- Модуль ВЧ-демпфування: Несправність: перенапруга 24 В'; 37052 'F37052 - Модуль ВЧ-демпфування: Помилка даних EEPROM'; 37056 'A37056 (F) - Модуль ВЧ-демпфування: Перегрів радіатора'; 37310 'A37310 (F) - Модуль ВЧ-дроселя: Перегрів'; 37311 'F37311 - Модуль ВЧ-дроселя: Перегрів радіатора'; 37312 'A37312 (F) - Модуль ВЧ-дроселя: Перегрів або несправність вентилятора'; 37313 'F37313 - Модуль ВЧ-дроселя: Перегрів або несправність вентилятора'; 37502 'A37502 (F) - Модуль ВЧ-демпфування: Напруга демпфування занадто висока'; 37800 'N37800 (F) - Модуль ВЧ-демпфування: Груповий сигнал'; 37801 'A37801 (F, N) - Модуль ВЧ-демпфування: Відсутній сигнал справності'; 37802 'F37802 (N, A) - Модуль ВЧ-демпфування: Переповнення часового кванта'; 37804 'F37804 (N, A) - Модуль ВЧ-демпфування: CRC'; 37805 'F37805 - Модуль ВЧ-демпфування: Некоректна контрольна сума EEPROM'; 37820 'F37820 - Модуль ВЧ-демпфування: Помилка телеграми'; 37835 'F37835 - Модуль ВЧ-демпфування: Помилка циклічної передачі даних'; 37836 'F37836 - Модуль ВЧ-демпфування: Помилка передавання даних DRIVE-CLiQ'; 37837 'F37837 - Модуль ВЧ-демпфування: Несправність компонента'; 37845 'F37845 - Модуль ВЧ-демпфування: Помилка циклічної передачі даних'; 37850 'F37850 - Модуль ВЧ-демпфування: Внутрішня програмна помилка'; 37851 'F37851 - Модуль ВЧ-демпфування (CU): Відсутній сигнал справності'; 37860 'F37860 - Модуль ВЧ-демпфування (CU): Помилка телеграми'; 37875 'F37875 - Модуль ВЧ-демпфування: Несправність напруги живлення'; 37885 'F37885 - Модуль ВЧ-демпфування (CU): Помилка циклічної передачі даних'; 37886 'F37886 - Модуль ВЧ-демпфування (CU): Помилка під час передавання даних DRIVE-CLiQ'; 37887 'F37887 - Модуль ВЧ-демпфування (CU): Несправність компонента'; 37895 'F37895 - Модуль ВЧ-демпфування (CU): Помилка почергової циклічної передачі даних'; 37896 'F37896 - Модуль ВЧ-демпфування (CU): Некоректні властивості компонента'; 37899 'F37899 (N, A) - Модуль ВЧ-демпфування: Невідома несправність'; 37903 'F37903 - Модуль ВЧ-демпфування: Виникла помилка I2C-шини'; 37950 'F37950 - Модуль ВЧ-демпфування: Внутрішня програмна помилка'; 37999 'A37999 (F, N) - Модуль ВЧ-демпфування: Невідоме аварійне повідомлення'; 40000 'F40000 - Несправність роз’єму DRIVE-CLiQ X100'; 40001 'F40001 - Несправність роз’єму DRIVE-CLiQ X101'; 40002 'F40002 - Несправність роз’єму DRIVE-CLiQ X102'; 40003 'F40003 - Несправність роз’єму DRIVE-CLiQ X103'; 40004 'F40004 - Несправність роз’єму DRIVE-CLiQ X104'; 40005 'F40005 - Несправність роз’єму DRIVE-CLiQ X105'; 40100 'A40100 - Аварійне повідомлення роз’єму DRIVE-CLiQ X100'; 40101 'A40101 - Аварійне повідомлення роз’єму DRIVE-CLiQ X101'; 40102 'A40102 - Аварійне повідомлення роз’єму DRIVE-CLiQ X102'; 40103 'A40103 - Аварійне повідомлення роз’єму DRIVE-CLiQ X103'; 40104 'A40104 - Аварійне повідомлення роз’єму DRIVE-CLiQ X104'; 40105 'A40105 - Аварійне повідомлення роз’єму DRIVE-CLiQ X105'; 40799 'F40799 - CX32: Перевищено налаштований час завершення передавання'; 40801 'F40801 - CX32 DRIVE-CLiQ: відсутній сигнал справності'; 40820 'F40820 - CX32 DRIVE-CLiQ: помилка телеграми'; 40825 'F40825 - CX32 DRIVE-CLiQ: Несправність напруги живлення'; 40835 'F40835 - CX32 DRIVE-CLiQ: помилка циклічної передачі даних'; 40836 'F40836 - CX32 DRIVE-CLiQ: помилка передавання даних DRIVE-CLiQ'; 40837 'F40837 - CX32 DRIVE-CLiQ: несправність компонента'; 40845 'F40845 - CX32 DRIVE-CLiQ: помилка циклічної передачі даних'; 40851 'F40851 - CX32 DRIVE-CLiQ (CU): відсутній сигнал справності'; 40860 'F40860 - CX32 DRIVE-CLiQ (CU): помилка телеграми'; 40875 'F40875 - CX32 DRIVE-CLiQ (CU): Несправність напруги живлення'; 40885 'F40885 - CX32 DRIVE-CLiQ (CU): помилка циклічної передачі даних'; 40886 'F40886 - CX32 DRIVE-CLiQ (CU): помилка під час передавання даних DRIVE-CLiQ'; 40887 'F40887 - CX32 DRIVE-CLiQ (CU): несправність компонента'; 40895 'F40895 - CX32 DRIVE-CLiQ (CU): помилка циклічної передачі даних'; 49150 'F49150 - Охолоджувальний агрегат: Виникла несправність'; 49151 'F49151 - Охолоджувальний агрегат: Провідність перевищила поріг несправності'; 49152 'F49152 - Охолоджувальний агрегат: Відсутній сигнал зворотного зв’язку команди ON'; 49153 'F49153 - Охолоджувальний агрегат: Витрата рідини занадто мала'; 49154 'F49154 (A) - Охолоджувальний агрегат: Виявлено витік рідини'; 49155 'F49155 - Охолоджувальний агрегат: Адаптер Power Stack: версія прошивки застаріла'; 49156 'F49156 - Охолоджувальний агрегат: Температура охолоджувальної рідини перевищила поріг несправності'; 49170 'A49170 - Охолоджувальний агрегат: Виникло аварійне повідомлення'; 49171 'A49171 (N) - Охолоджувальний агрегат: Провідність перевищила поріг аварійного повідомлення'; 49172 'A49172 - Охолоджувальний агрегат: Фактичне значення провідності некоректне'; 49173 'A49173 - Охолоджувальний агрегат: Температура охолоджувальної рідини перевищила поріг аварійного повідомлення'; 49200 'F49200 - Несправність групового сигналу збудження'; 49201 'A49201 (F) - Аварійне повідомлення групового сигналу збудження'; 49204 'A49204 (N) - Аварійне повідомлення про вимкнення збудження'; 49205 'A49205 - Збудження: некоректна параметризація безщіткового збуджувача'; 49920 'A49920 (F) - Спрацював захисний автомат головного кола'; 49921 'A49921 (F) - Спрацював захисний автомат резервного головного кола'; 49922 'A49922 (F) - Спрацював захисний автомат кола 24 В'; 49923 'A49923 (F) - Спрацював захисний автомат кола 24 В клемної колодки'; 49924 'A49924 (F) - Спрацював захисний автомат кола живлення силового модуля'; 49926 'A49926 (F) - Спрацював захисний автомат кола синхронізувальної напруги'; 49927 'A49927 (F) - Спрацював захисний автомат кола допоміжного вентилятора'; 49933 'A49933 (F) - Спрацював захисний автомат кола збудження 230 В AC'; 49934 'A49934 (F) - Спрацював захисний автомат вихідного кола охолоджувального агрегату 230 В AC'; 49935 'A49935 (F) - Спрацював захисний автомат кола 24 В соленоїдів дверей силового модуля'; 49936 'A49936 - Спрацював захисний автомат кола освітлення/розеток 230 В AC'; 49937 'A49937 (F) - UPS не готовий до роботи'; 49938 'A49938 (F) - Робота від батареї UPS'; 49939 'A49939 (F) - Батарею UPS розряджено'; 49940 'A49940 (F) - Спрацював захисний автомат кола живлення силового модуля 400 В'; 49941 'A49941 (F) - Спрацював захисний автомат антиконденсаційного обігріву'; 49942 'A49942 (F) - Спрацював захисний автомат кола живлення SITOP'; 49998 'A49998 - Виникла подія запуску реєстратора'; 50002 'A50002 (F) - COMM BOARD: аварійне повідомлення 2'; 50003 'A50003 (F) - COMM BOARD: аварійне повідомлення 3'; 50004 'A50004 (F) - COMM BOARD: аварійне повідомлення 4'; 50005 'A50005 (F) - COMM BOARD: аварійне повідомлення 5'; 50006 'A50006 (F) - COMM BOARD: аварійне повідомлення 6'; 50007 'A50007 (F) - COMM BOARD: аварійне повідомлення 7'; 50008 'A50008 (F) - COMM BOARD: аварійне повідомлення 8'; 50011 'A50011 (F) - EtherNetIP/COMM BOARD: помилка конфігурації'; 0 'Немає попередження'

text list "LiftUpStatus": 0 'Не має статусу'; 1 'Рухається вверх'; 2 'Рухається вниз'; 4 'Зупинено і Готовий до роботи (в середній зоні)'; 8 'Зупинено і НЕ готовий до роботи'; 16 'Аварія'; 32 'Зупинено у верхньому положенні'; 64 'Зупинено у нижньому положенні'

text list "TrolleyStatus": 1 'Рухається вперед'; 2 'Рухається назад'; 4 'Зупинено і Готовий до роботи'; 8 'Зупинено і НЕ готовий до роботи'; 16 'Аварія візка'; 32 'Зупинено у крайньому положенні Вперед'; 64 'Зупинено у крайньому положенні Назад'; 0 'Не має статусу'

text list "CraneStatus": 0 'Не має статусу'; 1 'Рухається вліво'; 2 'Рухається вправо'; 4 'Зупинено і Готовий до роботи'; 8 'Зупинено і НЕ готовий до роботи'; 16 'Аварія візка'; 32 'Зупинено у крайньому положенні Вліво'; 64 'Зупинено у крайньому положенні Вправо'

text list "LiftUpCondition": 0 'Очікується запуск калібровки'; 10 'Відпустіть всі кнопки керування / Відпустіть кнопки керування'; 20 'Натисніть кнопку «Підйом»'; 30 'Досягніть реперної точки 1K1'; 40 'Відпустіть кнопку «Підйом»'; 50 'Натисніть кноп. «Опускання», звільнить 1К1 та відпустіть кноп. / Звільніть 1K1 та відпустіть кнопку «Опускання»'; 60 'Відхід завершено'; 70 'Натисніть кнопку «Підйом»'; 80 'Повторно досягніть 1K1 та відпустіть кнопку / Повторно досягніть реперної точки 1K1'; 90 'Виконується Quick Stop'; 100 'Очікується повна зупинка привода, відпустіть кнопку "Підйом" / Очікується повна зупинка привода'; 110 'Запускається preset енкодера'; 120 'Очікується підтвердження preset енкодера / Очікується підтвердження preset'; 130 'Калібровка завершена'; 900 'Процедуру перервано'; 910 'Процедура завершена з помилкою'; 5 'Опустіться до звільнення 1К1 та відпустіть кнопку'

text list "LiftUpStepName": 0 'Калібровка неактивна'; 10 'Перевірка умов калібровки'; 20 'Очікування команди підйому'; 30 'Перший підхід до реперної точки'; 40 'Перше проходження 1K1'; 50 'Відхід нижче реперної точки'; 60 'Відхід завершено'; 70 'Очікування повторного підйому'; 80 'Повторний підхід до реперної точки'; 90 'Quick Stop'; 100 'Очікування зупинки привода'; 110 'Запуск preset енкодера'; 120 'Очікування завершення preset'; 130 'Калібровку успішно завершено'; 900 'Калібровку перервано'; 910 'Помилка калібровки'; 5 'Попередній відхід від реперної точки'

text list "TrolleyCondition": 0 'Очікується запуск калібровки'; 5 'Опустіться до звільнення 3К1 та відпустіть кнопку "Назад"'; 10 'Відпустіть всі кнопки керування / Відпустіть кнопки керування'; 20 'Натисніть кнопку «Підйом» / Натисніть кнопку «Вперед»'; 30 'Досягніть реперної точки 1K1 / Досягніть реперної точки 3K1'; 40 'Відпустіть кнопку «Підйом» / Відпустіть кнопку «Вперед»'; 50 'Звільніть 1K1 та відпустіть кнопку «Опускання» / Звільніть 3K1 та відпустіть кнопку «Назад»'; 60 'Відхід завершено'; 70 'Натисніть кнопку «Підйом» / Натисніть кнопку «Вперед»'; 80 'Повторно досягніть реперної точки 1K1 / Повторно досягніть 3K1 та відпустіть кнопку'; 90 'Виконується Quick Stop'; 100 'Очікується повна зупинка привода / Очікується повна зупинка привода, відпустіть кнопку "Вперед"'; 110 'Запускається preset енкодера'; 120 'Очікується підтвердження preset енкодера / Очікується підтвердження preset'; 130 'Калібровка завершена'; 900 'Процедуру перервано'; 910 'Процедура завершена з помилкою'

text list "TrolleyStepName": 0 'Калібровка неактивна'; 5 'Попередній відхід від реперної точки'; 10 'Перевірка умов калібровки'; 20 'Очікування команди підйому / Очікування команди руху вперед'; 30 'Перший підхід до реперної точки'; 40 'Перше проходження 1K1 / Перше проходження 3K1'; 50 'Відхід нижче реперної точки / Відхід назад від реперної точки'; 60 'Відхід завершено'; 70 'Очікування повторного підйому / Очікування повторного руху вперед'; 80 'Повторний підхід до реперної точки'; 90 'Quick Stop'; 100 'Очікування зупинки привода'; 110 'Запуск preset енкодера'; 120 'Очікування завершення preset'; 130 'Калібровку успішно завершено'; 900 'Калібровку перервано'; 910 'Помилка калібровки'

text list "CraneCondition": 0 'Очікується запуск калібровки'; 5 'Очікується звільнення 4К1 та відпустіть кнопку "Вправо"'; 10 'Відпустіть всі кнопки керування / Відпустіть кнопки керування'; 20 'Натисніть кнопку «Підйом» / Натисніть кнопку «Вліво»'; 30 'Досягніть реперної точки 1K1 / Досягніть реперної точки 4K1'; 40 'Відпустіть кнопку «Підйом» / Відпустіть кнопку «Вліво»'; 50 'Звільніть 1K1 та відпустіть кнопку «Опускання» / Звільніть 4K1 та відпустіть кнопку «Вправо»'; 60 'Відхід завершено'; 70 'Натисніть кнопку «Підйом» / Натисніть кнопку «Вліво»'; 80 'Повторно досягніть реперної точки 1K1 / Повторно досягніть 4K1 та відпустіть кнопку'; 90 'Виконується Quick Stop'; 100 'Очікується повна зупинка привода / Очікується повна зупинка обох приводів, відпустіть кнопку "Вліво"'; 110 'Запускається preset енкодера'; 120 'Очікується підтвердження preset / Очікується підтвердження preset обох енкодерів'; 130 'Калібровка завершена'; 900 'Процедуру перервано'; 910 'Процедура завершена з помилкою'

text list "CraneStepName": 0 'Калібровка неактивна'; 5 'Попередній відхід від реперної точки'; 10 'Перевірка умов калібровки'; 20 'Очікування команди підйому / Очікування команди руху вліво'; 30 'Перший підхід до реперної точки'; 40 'Перше проходження 1K1 / Перше проходження 4K1'; 50 'Відхід нижче реперної точки / Відхід вправо від реперної точки'; 60 'Відхід завершено'; 70 'Очікування повторного підйому / Очікування повторного руху вліво'; 80 'Повторний підхід до реперної точки'; 90 'Quick Stop'; 100 'Очікування зупинки привода / Очікування зупинки приводів'; 110 'Запуск preset енкодера / Запуск preset енкодерів'; 120 'Очікування завершення preset'; 130 'Калібровку успішно завершено'; 900 'Калібровку перервано'; 910 'Помилка калібровки'

Template "Template_1" 800x454
   Button "btnSettings" at 620,411 size 83x40; TextOff 'Exit'; PictureOn "ExitRuntime_TP700_Comfort_TR"; PictureOff "Navigates to System screens for TP700 Comfort 17.0.0.0"; Authorization "User administration"
      Appearance <- "Tag_ScreenNumber"
      on Release: ActivateScreen("90_Налаштування", 0)
   Button "btnKalibration" at 531,411 size 83x40; TextOff 'Калібровка'
      on Release: ActivateScreen("80_Калібровка", 0)
      Appearance <- "Tag_ScreenNumber"
   Button "btnDiagnostics" at 266,411 size 83x40; TextOff 'Діагностика'
      on Release: ActivateScreen("70_Діагностика", 0)
      Appearance <- "Tag_ScreenNumber"
   Button "btnArchive" at 443,411 size 83x40; TextOff 'Архіви'
      on Release: ActivateScreen("60_Архіви(1UZ1)", 0)
      Appearance <- "Tag_ScreenNumber"
   Button "btnAlarms" at 354,411 size 83x40; TextOff 'Аварії/ Регістрація'; TextOn 'Аварії'
      on Release: ActivateScreen("40_Аварії", 0)
      Appearance <- "Tag_ScreenNumber"
   Button "btnDrives" at 177,411 size 83x40; TextOff 'Привода'
      on Release: ActivateScreen("30_Drives(CU)", 0)
      Appearance <- "Tag_ScreenNumber"
   Button "btnDevices" at 89,411 size 83x40; TextOff 'Механізми'
      on Release: ActivateScreen("20_Механізми", 0)
      Appearance <- "Tag_ScreenNumber"
   Button "btnGeneralView" at 1,411 size 83x40; TextOff 'Головний екран'; PictureOff "NavigateHome_TP700_Comfort_TR"; PictureOn "NavigateHome_TP700_Comfort_TR"
      on Release: ActivateScreen("10_ГоловнийЕкран", 0)
      Appearance <- "Tag_ScreenNumber"
   DateTimeField "HmiScreenItemData" at 704,411 size 90x20
   DateTimeField "HmiScreenItemData_1" at 706,431 size 90x20

screen "90_Налаштування" 800x454, template "Template_1"
   on GenerateScreen: SetTag("Tag_ScreenNumber", 90)
   Button "HmiScreenItemData_2" at 36,133 size 190x50; TextOff 'Інформація о системі'; PictureOff "Navigates to System information for TP700 Comfort 17.0.0.0"; PictureOn "Navigates to System information for TP700 Comfort 17.0.0.0"
      on Release: ActivateScreen("92_ІнформацяіСистеми", 0)
   Button "HmiScreenItemData_3" at 36,192 size 190x50; TextOff 'Сервісні роботи'; PictureOff "Navigates to Different jobs for TP700 Comfort 17.0.0.0"; PictureOn "Navigates to Different jobs for TP700 Comfort 17.0.0.0"
      on Release: ActivateScreen("94_СервісніРоботи", 0)
   TextField "Text field_22" at 292,6 size 294x23; Text 'Головний екран налаштування'

screen "91_НалаштуванняЕкрану" 800x454, template "Template_1"
   on GenerateScreen: SetTag("Tag_ScreenNumber", 91)
   Button "Calibrate screen" at 36,115 size 190x50; TextOff 'Калібровка екрану'
      on Release: function_bc3e350c()
   Button "Clean screen" at 36,174 size 190x50; TextOff 'Очистка екрану'
      on Release: function_be740847(30)
   Button "Back" at 1,21 size 159x47; TextOff 'Назад'
      on Release: ActivateScreen("90_Налаштування", 10)
   TextField "Text field_22" at 292,6 size 213x23; Text 'Налаштування екрану'

screen "93_Адміністрування" 800x454, template "Template_1"
   on GenerateScreen: SetTag("Tag_ScreenNumber", 93)
   UserView "HmiScreenItemData20" at 1,69 size 796x304
   Button "Back" at 1,21 size 159x47; TextOff 'Назад'
      on Release: ActivateScreen("90_Налаштування", 10)
   TextField "Text field_22" at 292,6 size 296x23; Text 'Адіміністрування користувачів'

screen "92_ІнформацяіСистеми" 800x454, template "Template_1"
   on GenerateScreen: SetTag("Tag_ScreenNumber", 92)
   TextField "HmiScreenItemData_11" at 35,71 size 171x28; Text 'Типу ЛМІ:'
   TextField "HmiScreenItemData_10" at 241,71 size 524x28; Text 'TP700 Comfort 17.0.0.0'
   TextField "HmiScreenItemData_12" at 35,101 size 171x28; Text 'Версія:'
   TextField "HmiScreenItemData_13" at 35,131 size 171x28; Text 'З'єднання:'
   TextField "HmiScreenItemData_14" at 241,131 size 524x28; Text 'ETHERNET'
   TextField "HmiScreenItemData_15" at 35,161 size 171x28; Text 'ПЛК:'
   TextField "HmiScreenItemData_16" at 241,161 size 524x28; Text 'SIMATIC S7 1500'
   Button "Display version" at 241,101 size 524x28; TextOff 'Версія дісплею'
      on Release: function_febcb963(-1)
   Button "Back" at 1,21 size 159x47; TextOff 'Назад'
      on Release: ActivateScreen("90_Налаштування", 0)
   TextField "Text field_22" at 292,6 size 231x23; Text 'Інформація про систему'

screen "30_Drives(CU)" 800x454, template "Template_1"
   on GenerateScreen: SetTag("Tag_ScreenNumber", 30); SetTag("iVisibilityDevices", 0)
   Rectangle "rctCU320" at 7,79 size 98x34
      Visibility <- "Error"
   Rectangle "rct1UZ1" at 7,119 size 98x34
      Visibility <- "Error"
   Rectangle "rct4UZ1" at 7,199 size 98x34
      Visibility <- "Error"
   Rectangle "rct3UZ1" at 7,159 size 98x34
      Visibility <- "Error"
   Button "btn1UZ1" at 8,120 size 96x32; TextOff '1UZ1'
      on Release: ActivateScreen("31_Drives(1UZ1)", 0)
   Button "btn3UZ1" at 8,160 size 96x32; TextOff '3UZ1'
      on Release: ActivateScreen("32_Drives(3UZ1)", 0)
   Button "btn4UZ1" at 8,200 size 96x32; TextOff '4UZ1'
      on Release: ActivateScreen("33_Drives(4UZ1)", 0)
   Button "btnCU320" at 8,80 size 96x32; TextOff 'Модуль Кер. CU320 - 2PN'
   Rectangle "rct4UZ2" at 7,239 size 98x34
      Visibility <- "Error"
   Button "btn4UZ2" at 8,240 size 96x32; TextOff '4UZ2'
      on Release: ActivateScreen("34_Drives(4UZ2)", 0)
   Circle "Circle_1" at 130,54 size 16x16
      Visibility <- "iVisibilityDevices"
      Appearance <- "FaultAcknowledge"
   TextField "Text field_1" at 158,53 size 250x18; Text 'Квитування помилки'
      Visibility <- "iVisibilityDevices"
   Circle "Circle_2" at 130,74 size 16x16
      Visibility <- "iVisibilityDevices"
      Appearance <- "RemoteControlByPLC"
   TextField "Text field_2" at 158,73 size 250x18; Text 'Керування від PLC'
      Visibility <- "iVisibilityDevices"
   Circle "Circle_3" at 441,54 size 16x16
      Visibility <- "iVisibilityDevices"
      Appearance <- "ReadyToSwitchOn"
   TextField "Text field_5" at 469,53 size 250x18; Text 'CU готовий до вмикання / готовність'
      Visibility <- "iVisibilityDevices"
   Circle "Circle_4" at 441,74 size 16x16
      Visibility <- "iVisibilityDevices"
      Appearance <- "ReadyToOperate"
   TextField "Text field_6" at 469,73 size 250x18; Text 'CU готовий до роботи'
      Visibility <- "iVisibilityDevices"
   Circle "Circle_5" at 441,94 size 16x16
      Visibility <- "iVisibilityDevices"
      Appearance <- "OperationEnabled"
   TextField "Text field_7" at 469,93 size 250x18; Text 'Робота дозволена / стан ОК'
      Visibility <- "iVisibilityDevices"
   Circle "Circle_6" at 441,114 size 16x16
      Visibility <- "iVisibilityDevices"
      Appearance <- "FaultActive"
   TextField "Text field_8" at 469,113 size 250x18; Text 'Активна помилка CU'
      Visibility <- "iVisibilityDevices"
   Circle "Circle_7" at 441,134 size 16x16
      Visibility <- "iVisibilityDevices"
      Appearance <- "NoCoastStopActive"
   TextField "Text field_9" at 469,133 size 250x18; Text 'OFF2 не активний'
      Visibility <- "iVisibilityDevices"
   Circle "Circle_8" at 441,154 size 16x16
      Visibility <- "iVisibilityDevices"
      Appearance <- "NoQuickStopActive"
   TextField "Text field_10" at 469,153 size 250x18; Text 'OFF3 не активний'
      Visibility <- "iVisibilityDevices"
   Circle "Circle_9" at 441,174 size 16x16
      Visibility <- "iVisibilityDevices"
      Appearance <- "SwitchingOnInhibit"
   TextField "Text field_11" at 469,173 size 250x18; Text 'Заборона вмикання / блокування'
      Visibility <- "iVisibilityDevices"
   Circle "Circle_10" at 441,194 size 16x16
      Visibility <- "iVisibilityDevices"
      Appearance <- "WarningActive"
   TextField "Text field_12" at 469,193 size 250x18; Text 'Попередження'
      Visibility <- "iVisibilityDevices"
   Circle "Circle_11" at 441,214 size 16x16
      Visibility <- "iVisibilityDevices"
      Appearance <- "ControlRequested"
   TextField "Text field_13" at 469,213 size 250x18; Text 'Запит керування від PLC'
      Visibility <- "iVisibilityDevices"
   TextField "Text field_3" at 119,23 size 154x21; Text 'Слово керування:'
      Visibility <- "iVisibilityDevices"
   TextField "Text field_4" at 430,23 size 127x21; Text 'Слово статусу:'
      Visibility <- "iVisibilityDevices"

screen "40_Аварії" 800x454, template "Template_1"
   on GenerateScreen: SetTag("Tag_ScreenNumber", 40); SetTag("iVisibilityDevices", 0)
   AlarmView "alwContactor" at 119,29 size 675x370; ColumnTextDate 'Дата'; ColumnTextTime 'Час'; ColumnTextAlarmText 'Повідомлення'; ColumnTextAlarmState 'Обладнання'; AlarmLog "AlmVFD"
      Visibility <- "iVisibilityDevices"
   AlarmView "alwLiftUp" at 119,29 size 675x370; ColumnTextDate 'Дата'; ColumnTextTime 'Час'; ColumnTextAlarmText 'Повідомлення'; ColumnTextAlarmState 'Обладнання'; AlarmLog "AlmVFD"
      Visibility <- "iVisibilityDevices"
   AlarmView "alwTrolley" at 119,29 size 675x370; ColumnTextDate 'Дата'; ColumnTextTime 'Час'; ColumnTextAlarmText 'Повідомлення'; ColumnTextAlarmState 'Обладнання'; AlarmLog "AlmVFD"
      Visibility <- "iVisibilityDevices"
   AlarmView "alwCrane" at 119,29 size 675x370; ColumnTextDate 'Дата'; ColumnTextTime 'Час'; ColumnTextAlarmText 'Повідомлення'; ColumnTextAlarmState 'Обладнання'; AlarmLog "AlmVFD"
      Visibility <- "iVisibilityDevices"
   AlarmView "alwDiag" at 119,29 size 675x370; ColumnTextDate 'Дата'; ColumnTextTime 'Час'; ColumnTextAlarmText 'Повідомлення'; ColumnTextAlarmState 'Обладнання'; AlarmLog "AlmVFD"
      Visibility <- "iVisibilityDevices"
   Button "btnLiftUp" at 8,120 size 96x32; TextOff 'Механізм підйому'
      on Release: SetTag("iVisibilityDevices", 1)
      Appearance <- "iVisibilityDevices"
   Button "btnTrolley" at 8,160 size 96x32; TextOff 'Механізм візка'
      on Click: SetTag("iVisibilityDevices", 2)
      Appearance <- "iVisibilityDevices"
   Button "btnCrane" at 8,200 size 96x32; TextOff 'Механізм крану'
      on Release: SetTag("iVisibilityDevices", 3)
      Appearance <- "iVisibilityDevices"
   Button "btnContactor" at 8,80 size 96x32; TextOff 'Лінійний контактор'
      on Release: SetTag("iVisibilityDevices", 0)
      Appearance <- "iVisibilityDevices"
   Button "btnCrane_1" at 8,240 size 96x32; TextOff 'Діагностика'
      on Release: SetTag("iVisibilityDevices", 4)
      Appearance <- "iVisibilityDevices"
   Button "Button_1" at 8,367 size 96x32; TextOff 'Регістрація'; TextOn 'Діагностика'
      on Release: ActivateScreen("41_РегістраціяПодій", 0)
   TextField "Text field_1" at 425,5 size 63x23; Text 'Аварії'

screen "50_Trends(1UZ1)" 800x454, template "Template_1"
   on GenerateScreen: SetTag("Tag_ScreenNumber", 50); SetTag("iVisibilityDevices", 0)
   TrendView "trvCurrent" at 155,10 size 640x200
      Visibility <- "iVisibilityDevices"
   TrendView "trvMoment" at 155,208 size 640x200
      Visibility <- "iVisibilityDevices"
   TextField "txtCurrent" at 125,95 size 19x30; Text 'I ,А'
      Visibility <- "iVisibilityDevices"
   TextField "txtMoment" at 125,278 size 19x60; Text 'M , Н*м'
      Visibility <- "iVisibilityDevices"
   Button "btnLiftUp" at 8,120 size 96x32; TextOff '3UZ1'
      on Release: ActivateScreen("51_Trends(3UZ1)", 0)
   Button "btnTrolley" at 8,160 size 96x32; TextOff '4UZ1'
      on Release: ActivateScreen("52_Trends(4UZ1)", 0)
   Button "btnCrane" at 8,200 size 96x32; TextOff '4UZ2'
      on Release: ActivateScreen("53_Trends(4UZ2)", 0)
   Button "btnContactor" at 8,80 size 96x32; TextOff '1UZ1'
   Button "Button_1" at 8,319 size 96x32; TextOff 'Струм Момент'
      on Release: SetTag("iVisibilityDevices", 0)
      Appearance <- "iVisibilityDevices"
   Button "Button_2" at 8,356 size 96x32; TextOff 'Швидкості'
      on Release: SetTag("iVisibilityDevices", 1)
      Appearance <- "iVisibilityDevices"
   Button "Button_3" at 4,10 size 104x34; TextOff 'Діагностика / Діагностіка'; TextOn 'Діагностика'
      on Release: ActivateScreen("70_Діагностика", 0)
   TrendView "trvSpeed" at 155,10 size 640x200
      Visibility <- "iVisibilityDevices"
   TrendView "trvError" at 155,208 size 640x200
      Visibility <- "iVisibilityDevices"
   TextField "txtSpeed" at 108,84 size 19x53; Text 'W_set,'
      Visibility <- "iVisibilityDevices"
   TextField "txtError" at 125,259 size 19x98; Text 'W_err ,об/хв'
      Visibility <- "iVisibilityDevices"
   TextField "txtSpeed_1" at 120,82 size 19x57; Text 'W_real,'
      Visibility <- "iVisibilityDevices"
   TextField "txtSpeed_2" at 132,87 size 19x46; Text 'об/хв'
      Visibility <- "iVisibilityDevices"

screen "60_Архіви(1UZ1)" 800x454, template "Template_1"
   on GenerateScreen: SetTag("Tag_ScreenNumber", 60); SetTag("iVisibilityDevices", 0)
   Button "btnLiftUp" at 8,120 size 96x32; TextOff '3UZ1'
      on Release: ActivateScreen("61_Архіви(3UZ1)", 0)
   Button "btnTrolley" at 8,160 size 96x32; TextOff '4UZ1'
      on Release: ActivateScreen("62_Архіви(4UZ1)", 0)
   Button "btnCrane" at 8,200 size 96x32; TextOff '4UZ2'
      on Release: ActivateScreen("63_Архіви(4UZ2)", 0)
   Button "btnContactor" at 8,80 size 96x32; TextOff '1UZ1'
   Button "Button_1" at 8,319 size 96x32; TextOff 'Струм Момент'
      on Release: SetTag("iVisibilityDevices", 0)
      Appearance <- "iVisibilityDevices"
   Button "Button_2" at 8,356 size 96x32; TextOff 'Швидкості'
      on Release: SetTag("iVisibilityDevices", 1)
      Appearance <- "iVisibilityDevices"
   TrendView "trvCurrent" at 155,10 size 640x200
      Visibility <- "iVisibilityDevices"
   TrendView "trvMoment" at 155,208 size 640x200
      Visibility <- "iVisibilityDevices"
   TextField "txtCurrent" at 125,95 size 19x30; Text 'I ,А'
      Visibility <- "iVisibilityDevices"
   TextField "txtMoment" at 125,278 size 19x60; Text 'M , Н*м'
      Visibility <- "iVisibilityDevices"
   Button "btnCurrentDoubleBack" at 111,10 size 40x20; TextOff 'Text'; PictureOff "FB_2ArrowsLeft_Rectangular_Released_256c"; PictureOn "FB_2ArrowsLeft_Rectangular_Pressed_256c"
      Visibility <- "iVisibilityDevices"
      on Press: function_f26ff0ec("trvCurrent")
      on Release: function_f26ff0ec("trvCurrent")
   Button "btnCurrentOneBack" at 111,35 size 40x20; TextOff 'Text'; PictureOff "FB_ArrowLeft_Rectangular_Released_256c"; PictureOn "FB_ArrowLeft_Rectangular_Pressed_256c"
      Visibility <- "iVisibilityDevices"
      on Press: function_f26ff0ec("trvCurrent")
   Button "btnCurrentForward" at 111,149 size 40x20; TextOff 'Text'; PictureOff "FB_ArrowRight_Rectangular_Released_256c"; PictureOn "FB_ArrowRight_Rectangular_Pressed_256c"
      Visibility <- "iVisibilityDevices"
      on Press: function_c2ce674d("trvCurrent")
   Button "btnCurrentDoubleForward" at 111,174 size 40x20; TextOff 'Text'; PictureOff "FB_2ArrowsRight_Rectangular_Released_256c"; PictureOn "FB_2ArrowsRight_Rectangular_Pressed_256c"
      Visibility <- "iVisibilityDevices"
      on Press: function_c2ce674d("trvCurrent")
      on Release: function_c2ce674d("trvCurrent")
   Button "btnMomentDoubleBack" at 111,208 size 40x20; TextOff 'Text'; PictureOff "FB_2ArrowsLeft_Rectangular_Released_256c"; PictureOn "FB_2ArrowsLeft_Rectangular_Pressed_256c"
      Visibility <- "iVisibilityDevices"
      on Press: function_f26ff0ec("trvMoment")
      on Release: function_f26ff0ec("trvMoment")
   Button "btnMomentOneBack" at 111,233 size 40x20; TextOff 'Text'; PictureOff "FB_ArrowLeft_Rectangular_Released_256c"; PictureOn "FB_ArrowLeft_Rectangular_Pressed_256c"
      Visibility <- "iVisibilityDevices"
      on Press: function_f26ff0ec("trvMoment")
   Button "btnMomentOneForward" at 111,363 size 40x20; TextOff 'Text'; PictureOff "FB_ArrowRight_Rectangular_Released_256c"; PictureOn "FB_ArrowRight_Rectangular_Pressed_256c"
      Visibility <- "iVisibilityDevices"
      on Press: function_c2ce674d("trvMoment")
   Button "btnMomentDoubleForward" at 111,388 size 40x20; TextOff 'Text'; PictureOff "FB_2ArrowsRight_Rectangular_Released_256c"; PictureOn "FB_2ArrowsRight_Rectangular_Pressed_256c"
      Visibility <- "iVisibilityDevices"
      on Press: function_c2ce674d("trvMoment")
      on Release: function_c2ce674d("trvMoment")
   TrendView "trvSpeed" at 155,10 size 640x200
      Visibility <- "iVisibilityDevices"
   TrendView "trvError" at 155,208 size 640x200
      Visibility <- "iVisibilityDevices"
   TextField "txtSpeed" at 108,84 size 19x53; Text 'W_set,'
      Visibility <- "iVisibilityDevices"
   TextField "txtError" at 125,259 size 19x98; Text 'W_err ,об/хв'
      Visibility <- "iVisibilityDevices"
   TextField "txtSpeed_1" at 120,82 size 19x57; Text 'W_real,'
      Visibility <- "iVisibilityDevices"
   TextField "txtSpeed_2" at 132,87 size 19x46; Text 'об/хв'
      Visibility <- "iVisibilityDevices"
   Button "btnSpeedDoubleBack" at 111,10 size 40x20; TextOff 'Text'; PictureOff "FB_2ArrowsLeft_Rectangular_Released_256c"; PictureOn "FB_2ArrowsLeft_Rectangular_Pressed_256c"
      on Press: function_f26ff0ec("trvSpeed")
      on Release: function_f26ff0ec("trvSpeed")
      Visibility <- "iVisibilityDevices"
   Button "btnSpeedOneBack" at 111,35 size 40x20; TextOff 'Text'; PictureOff "FB_ArrowLeft_Rectangular_Released_256c"; PictureOn "FB_ArrowLeft_Rectangular_Pressed_256c"
      on Press: function_f26ff0ec("trvSpeed")
      Visibility <- "iVisibilityDevices"
   Button "btnSpeedForward" at 111,149 size 40x20; TextOff 'Text'; PictureOff "FB_ArrowRight_Rectangular_Released_256c"; PictureOn "FB_ArrowRight_Rectangular_Pressed_256c"
      on Press: function_c2ce674d("trvSpeed")
      Visibility <- "iVisibilityDevices"
   Button "btnSpeedDoubleForward" at 111,174 size 40x20; TextOff 'Text'; PictureOff "FB_2ArrowsRight_Rectangular_Released_256c"; PictureOn "FB_2ArrowsRight_Rectangular_Pressed_256c"
      on Press: function_c2ce674d("trvSpeed")
      on Release: function_c2ce674d("trvSpeed")
      Visibility <- "iVisibilityDevices"
   Button "btnErrorDoubleBack" at 111,208 size 40x20; TextOff 'Text'; PictureOff "FB_2ArrowsLeft_Rectangular_Released_256c"; PictureOn "FB_2ArrowsLeft_Rectangular_Pressed_256c"
      on Press: function_f26ff0ec("trvError")
      on Release: function_f26ff0ec("trvError")
      Visibility <- "iVisibilityDevices"
   Button "btnErrorOneBack" at 111,233 size 40x20; TextOff 'Text'; PictureOff "FB_ArrowLeft_Rectangular_Released_256c"; PictureOn "FB_ArrowLeft_Rectangular_Pressed_256c"
      on Press: function_f26ff0ec("trvError")
      Visibility <- "iVisibilityDevices"
   Button "btnErrorOneForward" at 111,363 size 40x20; TextOff 'Text'; PictureOff "FB_ArrowRight_Rectangular_Released_256c"; PictureOn "FB_ArrowRight_Rectangular_Pressed_256c"
      on Press: function_c2ce674d("trvError")
      Visibility <- "iVisibilityDevices"
   Button "btnErrorDoubleForward" at 111,388 size 40x20; TextOff 'Text'; PictureOff "FB_2ArrowsRight_Rectangular_Released_256c"; PictureOn "FB_2ArrowsRight_Rectangular_Pressed_256c"
      on Press: function_c2ce674d("trvError")
      on Release: function_c2ce674d("trvError")
      Visibility <- "iVisibilityDevices"

screen "94_СервісніРоботи" 800x454, template "Template_1"
   on GenerateScreen: SetTag("Tag_ScreenNumber", 94)
   Button "Stop Runtime" at 31,83 size 159x47; TextOff 'Стоп РТ'
      on Release: StopRuntime(0)
   Button "Back" at 1,21 size 159x47; TextOff 'Назад'
      on Release: ActivateScreen("90_Налаштування", 10)
   Button "btnStopLog" at 31,163 size 159x47; TextOff 'Стоп Логінг'
      on Release: "StopLog"()
      ObjectEnable <- "iStep"
   Button "btnStartLog" at 31,348 size 159x47; TextOff 'Старт Логінг'
      on Release: "StartLog"()
      ObjectEnable <- "iStep"
   Button "btnCopyLog" at 31,255 size 159x47; TextOff 'Старт Логінг / Копі Лог'; TextOn 'Старт Логінг'
      on Release: "CopyLogs"()
      ObjectEnable <- "iStep"
   TextField "Text field_22" at 292,6 size 153x23; Text 'Сервісні роботи'
   TextField "Text field_1" at 201,214 size 330x130; Text 'Перенос логів виконується у наступній черзі 1) Стоп Логінг - закриття та зупинка логів 2) Копі Лог - копіювання логів до USB 3) Старт Логінг - відкриття та запуск логів Номер кроку'
   Line "Line_1" at 111,214 size 0x36
      Visibility <- "iStep"
   Line "Line_2" at 111,308 size 0x36
      Visibility <- "iStep"

screen "71_A1.2(DI32)_1" 800x454, template "Template_1"
   on GenerateScreen: SetTag("iVisibilityA1.2", 0); SetTag("Tag_ScreenNumber", 71)
   ScreenModuleView "fcptDI0.0" at 117,32 size 680x18; ScreenModuleType ""
      Guid_{11997190-10951} <- "HMI_DB_IO_Tags_InCnf_DigIn_0_0"
   ScreenModuleView "fcptDI0.1" at 117,55 size 680x18; ScreenModuleType ""
      Guid_{11997190-10951} <- "HMI_DB_IO_Tags_InCnf_DigIn_0_1"
   ScreenModuleView "fcptDI0.2" at 117,78 size 680x18; ScreenModuleType ""
      Guid_{11997190-10951} <- "HMI_DB_IO_Tags_InCnf_DigIn_0_2"
   ScreenModuleView "fcptDI0.3" at 117,102 size 680x18; ScreenModuleType ""
      Guid_{11997190-10951} <- "HMI_DB_IO_Tags_InCnf_DigIn_0_3"
   ScreenModuleView "fcptDI0.4" at 117,125 size 680x18; ScreenModuleType ""
      Guid_{11997190-10951} <- "HMI_DB_IO_Tags_InCnf_DigIn_0_4"
   ScreenModuleView "fcptDI0.5" at 117,148 size 680x18; ScreenModuleType ""
      Guid_{11997190-10951} <- "HMI_DB_IO_Tags_InCnf_DigIn_0_5"
   ScreenModuleView "fcptDI0.6" at 117,172 size 680x18; ScreenModuleType ""
      Guid_{11997190-10951} <- "HMI_DB_IO_Tags_InCnf_DigIn_0_6"
   ScreenModuleView "fcptDI0.7" at 117,195 size 680x18; ScreenModuleType ""
      Guid_{11997190-10951} <- "HMI_DB_IO_Tags_InCnf_DigIn_0_7"
   ScreenModuleView "fcptDI1.0" at 117,218 size 680x18; ScreenModuleType ""
      Guid_{11997190-10951} <- "HMI_DB_IO_Tags_InCnf_DigIn_1_0"
   ScreenModuleView "fcptDI1.1" at 117,242 size 680x18; ScreenModuleType ""
      Guid_{11997190-10951} <- "HMI_DB_IO_Tags_InCnf_DigIn_1_1"
   ScreenModuleView "fcptDI1.2" at 117,265 size 680x18; ScreenModuleType ""
      Guid_{11997190-10951} <- "HMI_DB_IO_Tags_InCnf_DigIn_1_2"
   ScreenModuleView "fcptDI1.3" at 117,288 size 680x18; ScreenModuleType ""
      Guid_{11997190-10951} <- "HMI_DB_IO_Tags_InCnf_DigIn_1_3"
   ScreenModuleView "fcptDI1.4" at 117,312 size 680x18; ScreenModuleType ""
      Guid_{11997190-10951} <- "HMI_DB_IO_Tags_InCnf_DigIn_1_4"
   ScreenModuleView "fcptDI1.5" at 117,335 size 680x18; ScreenModuleType ""
      Guid_{11997190-10951} <- "HMI_DB_IO_Tags_InCnf_DigIn_1_5"
   ScreenModuleView "fcptDI1.6" at 117,358 size 680x18; ScreenModuleType ""
      Guid_{11997190-10951} <- "HMI_DB_IO_Tags_InCnf_DigIn_1_6"
   ScreenModuleView "fcptDI1.7" at 117,382 size 680x18; ScreenModuleType ""
      Guid_{11997190-10951} <- "HMI_DB_IO_Tags_InCnf_DigIn_1_7"
   Button "Button_2" at 8,96 size 96x32; TextOff 'DI0.0_DI1.7'
      Appearance <- "iVisibilityA1.2"
   Button "Button_3" at 8,159 size 96x32; TextOff 'DI2.0_DI3.7'
      on Press: SetTag("iVisibilityA1.2", 1); ActivateScreen("72_A1.2(DI32)_2", 0)
      Appearance <- "iVisibilityA1.2"
   TextField "Text field_1" at 282,6 size 350x23; Text 'Стан діскретних входів DI0.0 - DI1.7'

screen "72_A1.2(DI32)_2" 800x454, template "Template_1"
   on GenerateScreen: SetTag("Tag_ScreenNumber", 72)
   ScreenModuleView "fcptDI2.0" at 117,32 size 680x18; ScreenModuleType ""
      Guid_{11997190-10951} <- "HMI_DB_IO_Tags_InCnf_DigIn_2_0"
   ScreenModuleView "fcptDI2.1" at 117,55 size 680x18; ScreenModuleType ""
      Guid_{11997190-10951} <- "HMI_DB_IO_Tags_InCnf_DigIn_2_1"
   ScreenModuleView "fcptDI2.2" at 117,78 size 680x18; ScreenModuleType ""
      Guid_{11997190-10951} <- "HMI_DB_IO_Tags_InCnf_DigIn_2_2"
   ScreenModuleView "fcptDI2.3" at 117,102 size 680x18; ScreenModuleType ""
      Guid_{11997190-10951} <- "HMI_DB_IO_Tags_InCnf_DigIn_2_3"
   ScreenModuleView "fcptDI2.4" at 117,125 size 680x18; ScreenModuleType ""
      Guid_{11997190-10951} <- "HMI_DB_IO_Tags_InCnf_DigIn_2_4"
   ScreenModuleView "fcptDI2.5" at 117,148 size 680x18; ScreenModuleType ""
      Guid_{11997190-10951} <- "HMI_DB_IO_Tags_InCnf_DigIn_2_5"
   ScreenModuleView "fcptDI2.6" at 117,172 size 680x18; ScreenModuleType ""
      Guid_{11997190-10951} <- "HMI_DB_IO_Tags_InCnf_DigIn_2_6"
   ScreenModuleView "fcptDI2.7" at 117,195 size 680x18; ScreenModuleType ""
      Guid_{11997190-10951} <- "HMI_DB_IO_Tags_InCnf_DigIn_2_7"
   ScreenModuleView "fcptDI3.0" at 117,218 size 680x18; ScreenModuleType ""
      Guid_{11997190-10951} <- "HMI_DB_IO_Tags_InCnf_DigIn_3_0"
   ScreenModuleView "fcptDI3.1" at 117,242 size 680x18; ScreenModuleType ""
      Guid_{11997190-10951} <- "HMI_DB_IO_Tags_InCnf_DigIn_3_1"
   ScreenModuleView "fcptDI3.2" at 117,265 size 680x18; ScreenModuleType ""
      Guid_{11997190-10951} <- "HMI_DB_IO_Tags_InCnf_DigIn_3_2"
   ScreenModuleView "fcptDI3.3" at 117,288 size 680x18; ScreenModuleType ""
      Guid_{11997190-10951} <- "HMI_DB_IO_Tags_InCnf_DigIn_3_3"
   ScreenModuleView "fcptDI3.4" at 117,312 size 680x18; ScreenModuleType ""
      Guid_{11997190-10951} <- "HMI_DB_IO_Tags_InCnf_DigIn_3_4"
   ScreenModuleView "fcptDI3.5" at 117,335 size 680x18; ScreenModuleType ""
      Guid_{11997190-10951} <- "HMI_DB_IO_Tags_InCnf_DigIn_3_5"
   ScreenModuleView "fcptDI3.6" at 117,358 size 680x18; ScreenModuleType ""
      Guid_{11997190-10951} <- "HMI_DB_IO_Tags_InCnf_DigIn_3_6"
   ScreenModuleView "fcptDI3.7" at 117,382 size 680x18; ScreenModuleType ""
      Guid_{11997190-10951} <- "HMI_DB_IO_Tags_InCnf_DigIn_3_7"
   Button "Button_2" at 8,96 size 96x32; TextOff 'DI0.0_DI1.7'
      on Press: SetTag("iVisibilityA1.2", 0); ActivateScreen("71_A1.2(DI32)_1", 0)
      Appearance <- "iVisibilityA1.2"
   Button "Button_3" at 8,159 size 96x32; TextOff 'DI2.0_DI3.7'
      Appearance <- "iVisibilityA1.2"
   TextField "Text field_1" at 282,6 size 350x23; Text 'Стан діскретних входів DI2.0 - DI3.7'

screen "73_A1.3(DI32)_1" 800x454, template "Template_1"
   on GenerateScreen: SetTag("iVisibilityA1.3", 0); SetTag("Tag_ScreenNumber", 73)
   ScreenModuleView "fcptDI4.0" at 117,32 size 680x18; ScreenModuleType ""
      Guid_{11997190-10951} <- "HMI_DB_IO_Tags_InCnf_DigIn_4_0"
   ScreenModuleView "fcptDI4.1" at 117,55 size 680x18; ScreenModuleType ""
      Guid_{11997190-10951} <- "HMI_DB_IO_Tags_InCnf_DigIn_4_1"
   ScreenModuleView "fcptDI4.2" at 117,78 size 680x18; ScreenModuleType ""
      Guid_{11997190-10951} <- "HMI_DB_IO_Tags_InCnf_DigIn_4_2"
   ScreenModuleView "fcptDI4.3" at 117,102 size 680x18; ScreenModuleType ""
      Guid_{11997190-10951} <- "HMI_DB_IO_Tags_InCnf_DigIn_4_3"
   ScreenModuleView "fcptDI4.4" at 117,125 size 680x18; ScreenModuleType ""
      Guid_{11997190-10951} <- "HMI_DB_IO_Tags_InCnf_DigIn_4_4"
   ScreenModuleView "fcptDI4.5" at 117,148 size 680x18; ScreenModuleType ""
      Guid_{11997190-10951} <- "HMI_DB_IO_Tags_InCnf_DigIn_4_5"
   ScreenModuleView "fcptDI4.6" at 117,172 size 680x18; ScreenModuleType ""
      Guid_{11997190-10951} <- "HMI_DB_IO_Tags_InCnf_DigIn_4_6"
   ScreenModuleView "fcptDI4.7" at 117,195 size 680x18; ScreenModuleType ""
      Guid_{11997190-10951} <- "HMI_DB_IO_Tags_InCnf_DigIn_4_7"
   ScreenModuleView "fcptDI5.0" at 117,218 size 680x18; ScreenModuleType ""
      Guid_{11997190-10951} <- "HMI_DB_IO_Tags_InCnf_DigIn_5_0"
   ScreenModuleView "fcptDI5.1" at 117,242 size 680x18; ScreenModuleType ""
      Guid_{11997190-10951} <- "HMI_DB_IO_Tags_InCnf_DigIn_5_1"
   ScreenModuleView "fcptDI5.2" at 117,265 size 680x18; ScreenModuleType ""
      Guid_{11997190-10951} <- "HMI_DB_IO_Tags_InCnf_DigIn_5_2"
   ScreenModuleView "fcptDI5.3" at 117,288 size 680x18; ScreenModuleType ""
      Guid_{11997190-10951} <- "HMI_DB_IO_Tags_InCnf_DigIn_5_3"
   ScreenModuleView "fcptDI5.4" at 117,312 size 680x18; ScreenModuleType ""
      Guid_{11997190-10951} <- "HMI_DB_IO_Tags_InCnf_DigIn_5_4"
   ScreenModuleView "fcptDI5.5" at 117,335 size 680x18; ScreenModuleType ""
      Guid_{11997190-10951} <- "HMI_DB_IO_Tags_InCnf_DigIn_5_5"
   ScreenModuleView "fcptDI5.6" at 117,358 size 680x18; ScreenModuleType ""
      Guid_{11997190-10951} <- "HMI_DB_IO_Tags_InCnf_DigIn_5_6"
   ScreenModuleView "fcptDI5.7" at 117,382 size 680x18; ScreenModuleType ""
      Guid_{11997190-10951} <- "HMI_DB_IO_Tags_InCnf_DigIn_5_7"
   Button "Button_2" at 8,96 size 96x32; TextOff 'DI4.0_DI5.7'
      Appearance <- "iVisibilityA1.3"
   Button "Button_3" at 8,159 size 96x32; TextOff 'DI6.0_DI7.7'
      on Press: SetTag("iVisibilityA1.3", 1); ActivateScreen("74_A1.3(DI32)_2", 0)
      Appearance <- "iVisibilityA1.3"
   TextField "Text field_1" at 282,6 size 350x23; Text 'Стан діскретних входів DI4.0 - DI5.7'

screen "74_A1.3(DI32)_2" 800x454, template "Template_1"
   on GenerateScreen: SetTag("Tag_ScreenNumber", 74)
   ScreenModuleView "fcptDI6.0" at 117,32 size 680x18; ScreenModuleType ""
      Guid_{11997190-10951} <- "HMI_DB_IO_Tags_InCnf_DigIn_6_0"
   ScreenModuleView "fcptDI6.1" at 117,55 size 680x18; ScreenModuleType ""
      Guid_{11997190-10951} <- "HMI_DB_IO_Tags_InCnf_DigIn_6_1"
   ScreenModuleView "fcptDI6.2" at 117,78 size 680x18; ScreenModuleType ""
      Guid_{11997190-10951} <- "HMI_DB_IO_Tags_InCnf_DigIn_6_2"
   ScreenModuleView "fcptDI6.3" at 117,102 size 680x18; ScreenModuleType ""
      Guid_{11997190-10951} <- "HMI_DB_IO_Tags_InCnf_DigIn_6_3"
   ScreenModuleView "fcptDI6.4" at 117,125 size 680x18; ScreenModuleType ""
      Guid_{11997190-10951} <- "HMI_DB_IO_Tags_InCnf_DigIn_6_4"
   ScreenModuleView "fcptDI6.5" at 117,148 size 680x18; ScreenModuleType ""
      Guid_{11997190-10951} <- "HMI_DB_IO_Tags_InCnf_DigIn_6_5"
   ScreenModuleView "fcptDI6.6" at 117,172 size 680x18; ScreenModuleType ""
      Guid_{11997190-10951} <- "HMI_DB_IO_Tags_InCnf_DigIn_6_6"
   ScreenModuleView "fcptDI6.7" at 117,195 size 680x18; ScreenModuleType ""
      Guid_{11997190-10951} <- "HMI_DB_IO_Tags_InCnf_DigIn_6_7"
   ScreenModuleView "fcptDI7.0" at 117,218 size 680x18; ScreenModuleType ""
      Guid_{11997190-10951} <- "HMI_DB_IO_Tags_InCnf_DigIn_7_0"
   ScreenModuleView "fcptDI7.1" at 117,242 size 680x18; ScreenModuleType ""
      Guid_{11997190-10951} <- "HMI_DB_IO_Tags_InCnf_DigIn_7_1"
   ScreenModuleView "fcptDI7.2" at 117,265 size 680x18; ScreenModuleType ""
      Guid_{11997190-10951} <- "HMI_DB_IO_Tags_InCnf_DigIn_7_2"
   ScreenModuleView "fcptDI7.3" at 117,288 size 680x18; ScreenModuleType ""
      Guid_{11997190-10951} <- "HMI_DB_IO_Tags_InCnf_DigIn_7_3"
   ScreenModuleView "fcptDI7.4" at 117,312 size 680x18; ScreenModuleType ""
      Guid_{11997190-10951} <- "HMI_DB_IO_Tags_InCnf_DigIn_7_4"
   ScreenModuleView "fcptDI7.5" at 117,335 size 680x18; ScreenModuleType ""
      Guid_{11997190-10951} <- "HMI_DB_IO_Tags_InCnf_DigIn_7_5"
   ScreenModuleView "fcptDI7.6" at 117,358 size 680x18; ScreenModuleType ""
      Guid_{11997190-10951} <- "HMI_DB_IO_Tags_InCnf_DigIn_7_6"
   ScreenModuleView "fcptDI7.7" at 117,382 size 680x18; ScreenModuleType ""
      Guid_{11997190-10951} <- "HMI_DB_IO_Tags_InCnf_DigIn_7_7"
   Button "Button_2" at 8,96 size 96x32; TextOff 'DI6.0_DI7.7'
      on Press: SetTag("iVisibilityA1.3", 0); ActivateScreen("73_A1.3(DI32)_1", 0)
      Appearance <- "iVisibilityA1.3"
   Button "Button_3" at 8,159 size 96x32; TextOff 'DI6.0_DI7.7 / DI2.0_DI3.7'; TextOn 'DI2.0_DI3.7'
      Appearance <- "iVisibilityA1.3"
   TextField "Text field_1" at 282,6 size 350x23; Text 'Стан діскретних входів DI6.0 - DI7.7'

screen "75_A1.5(DQ16)" 800x454, template "Template_1"
   on GenerateScreen: SetTag("Tag_ScreenNumber", 75)
   ScreenModuleView "fcptDO0.0" at 117,32 size 680x18; ScreenModuleType ""
      Guid_{11997190-10951} <- "HMI_DB_IO_Tags_OutCfg_DigOut_0_0"
   ScreenModuleView "fcptDO1.7" at 117,382 size 680x18; ScreenModuleType ""
      Guid_{11997190-10951} <- "HMI_DB_IO_Tags_OutCfg_DigOut_1_7"
   ScreenModuleView "fcptDO0.1" at 117,55 size 680x18; ScreenModuleType ""
      Guid_{11997190-10951} <- "HMI_DB_IO_Tags_OutCfg_DigOut_0_1"
   ScreenModuleView "fcptDO0.2" at 117,78 size 680x18; ScreenModuleType ""
      Guid_{11997190-10951} <- "HMI_DB_IO_Tags_OutCfg_DigOut_0_2"
   ScreenModuleView "fcptDO0.4" at 117,125 size 680x18; ScreenModuleType ""
      Guid_{11997190-10951} <- "HMI_DB_IO_Tags_OutCfg_DigOut_0_4"
   ScreenModuleView "fcptDO0.5" at 117,148 size 680x18; ScreenModuleType ""
      Guid_{11997190-10951} <- "HMI_DB_IO_Tags_OutCfg_DigOut_0_5"
   ScreenModuleView "fcptDO0.6" at 117,172 size 680x18; ScreenModuleType ""
      Guid_{11997190-10951} <- "HMI_DB_IO_Tags_OutCfg_DigOut_0_6"
   ScreenModuleView "fcptDO0.7" at 117,195 size 680x18; ScreenModuleType ""
      Guid_{11997190-10951} <- "HMI_DB_IO_Tags_OutCfg_DigOut_0_7"
   ScreenModuleView "fcptDO1.0" at 117,218 size 680x18; ScreenModuleType ""
      Guid_{11997190-10951} <- "HMI_DB_IO_Tags_OutCfg_DigOut_1_0"
   ScreenModuleView "fcptDO1.1" at 117,242 size 680x18; ScreenModuleType ""
      Guid_{11997190-10951} <- "HMI_DB_IO_Tags_OutCfg_DigOut_1_1"
   ScreenModuleView "fcptDO1.2" at 117,265 size 680x18; ScreenModuleType ""
      Guid_{11997190-10951} <- "HMI_DB_IO_Tags_OutCfg_DigOut_1_2"
   ScreenModuleView "fcptDO1.3" at 117,288 size 680x18; ScreenModuleType ""
      Guid_{11997190-10951} <- "HMI_DB_IO_Tags_OutCfg_DigOut_1_3"
   ScreenModuleView "fcptDO1.4" at 117,312 size 680x18; ScreenModuleType ""
      Guid_{11997190-10951} <- "HMI_DB_IO_Tags_OutCfg_DigOut_1_4"
   ScreenModuleView "fcptDO1.5" at 117,335 size 680x18; ScreenModuleType ""
      Guid_{11997190-10951} <- "HMI_DB_IO_Tags_OutCfg_DigOut_1_5"
   ScreenModuleView "fcptDO0.3" at 117,102 size 680x18; ScreenModuleType ""
      Guid_{11997190-10951} <- "HMI_DB_IO_Tags_OutCfg_DigOut_0_3"
   ScreenModuleView "fcptDO1.6" at 117,358 size 680x18; ScreenModuleType ""
      Guid_{11997190-10951} <- "HMI_DB_IO_Tags_OutCfg_DigOut_1_6"
   TextField "Text field_1" at 282,6 size 371x23; Text 'Стан діскретних виходів DQ0.0 - DQ1.7'

screen "76_A1.4(IW8)" 800x454, template "Template_1"
   on GenerateScreen: SetTag("Tag_ScreenNumber", 76)
   ScreenModuleView "fcptAI18" at 117,32 size 580x18; ScreenModuleType ""
      Guid_{11997190-10951} <- "HMI_DB_IO_Tags_InAnCfg_AnIn_0"
   ScreenModuleView "fcptAI20" at 117,77 size 580x18; ScreenModuleType ""
      Guid_{11997190-10951} <- "HMI_DB_IO_Tags_InAnCfg_AnIn_1"
   ScreenModuleView "fcptAI22" at 117,122 size 580x18; ScreenModuleType ""
      Guid_{11997190-10951} <- "HMI_DB_IO_Tags_InAnCfg_AnIn_2"
   ScreenModuleView "fcptAI24" at 117,167 size 580x18; ScreenModuleType ""
      Guid_{11997190-10951} <- "HMI_DB_IO_Tags_InAnCfg_AnIn_3"
   ScreenModuleView "fcptAI26" at 117,212 size 580x18; ScreenModuleType ""
      Guid_{11997190-10951} <- "HMI_DB_IO_Tags_InAnCfg_AnIn_4"
   ScreenModuleView "fcptAI28" at 117,257 size 580x18; ScreenModuleType ""
      Guid_{11997190-10951} <- "HMI_DB_IO_Tags_InAnCfg_AnIn_5"
   ScreenModuleView "fcptAI30" at 117,302 size 580x18; ScreenModuleType ""
      Guid_{11997190-10951} <- "HMI_DB_IO_Tags_InAnCfg_AnIn_6"
   ScreenModuleView "fcptAI32" at 117,347 size 580x18; ScreenModuleType ""
      Guid_{11997190-10951} <- "HMI_DB_IO_Tags_InAnCfg_AnIn_7"
   TextField "Text field_1" at 282,6 size 368x23; Text 'Стан аналоговмх входів AIW8 - AIW22'

screen "77_1BR" 800x454, template "Template_1"
   on GenerateScreen: SetTag("Tag_ScreenNumber", 77)
   TextField "Text field_1" at 17,28 size 250x21; Text 'Слово керування енкодером:'
   Circle "Circle_1" at 28,55 size 16x16
      Appearance <- "STW2_ENC"
   Circle "Circle_2" at 28,75 size 16x16
      Appearance <- "ZSW2_ENC"
   Circle "Circle_3" at 28,95 size 16x16
      Appearance <- "STW2_ENC"
   TextField "Text field_3" at 56,54 size 231x18; Text 'Трігер на калібровку енкодера'
   TextField "Text field_4" at 56,74 size 154x18; Text 'Квитування помилки'
   TextField "Text field_5" at 56,94 size 123x18; Text 'Контроль з PLC'
   IOField "I/O field_1" at 16,115 size 40x20; FormatPattern FFFF
      ProcessValue <- "STW2_ENC"
   TextField "Text field_6" at 56,115 size 248x18; Text 'Сигнал працездатності енкодера'
   TextField "Text field_12" at 403,28 size 210x21; Text 'Слово статусу енкодера:'
   Circle "Circle_9" at 414,55 size 16x16
      Appearance <- "ZSW2_ENC"
   TextField "Text field_14" at 442,54 size 350x18; Text 'Підтвердження встановлення нового значення'
   Circle "Circle_10" at 414,75 size 16x16
      Appearance <- "ZSW2_ENC"
   TextField "Text field_15" at 442,74 size 234x18; Text 'Фактичне положення є дійсним'
   Circle "Circle_11" at 414,95 size 16x16
      Appearance <- "ZSW2_ENC"
   TextField "Text field_16" at 442,94 size 228x18; Text 'Фактична швидкість є дійсною'
   Circle "Circle_12" at 414,115 size 16x16
      Appearance <- "ZSW2_ENC"
   TextField "Text field_17" at 442,114 size 129x18; Text 'Помилка активна'
   Circle "Circle_13" at 414,135 size 16x16
      Appearance <- "ZSW2_ENC"
   TextField "Text field_18" at 442,134 size 176x18; Text 'Попередження активне'
   Circle "Circle_14" at 414,155 size 16x16
      Appearance <- "ZSW2_ENC"
   TextField "Text field_19" at 442,154 size 145x18; Text 'Запит на перевірку'
   TextField "Text field_20" at 442,174 size 248x18; Text 'Сигнал працездатності енкодера'
   IOField "I/O field_2" at 402,173 size 40x20; FormatPattern FFFF
      ProcessValue <- "ZSW2_ENC"
   IOField "I/O field_3" at 148,364 size 70x20; FormatPattern s9999999999
      ProcessValue <- "RawPosition"
   TextField "Text field_26" at 28,363 size 107x21; Text 'Положення:'
   IOField "I/O field_4" at 534,364 size 70x20; FormatPattern s9999999999
      ProcessValue <- "RawVelocity"
   TextField "Text field_27" at 414,363 size 97x21; Text 'Швидкість:'
   Circle "Circle_4" at 28,222 size 16x16
      Appearance <- "EncoderLifeValid"
   TextField "Text field_2" at 56,221 size 228x18; Text 'Sign-of-life енкодера валідний'
   Circle "Circle_5" at 28,242 size 16x16
      Appearance <- "EncoderReady"
   TextField "Text field_7" at 56,241 size 325x18; Text 'Енкодер готовий для використання в логіці'
   Circle "Circle_6" at 28,262 size 16x16
      Appearance <- "CommunicationFault"
   TextField "Text field_8" at 56,261 size 288x18; Text 'Загальна помилка обміну з енкодером'
   Circle "Circle_7" at 28,282 size 16x16
      Appearance <- "PresetBusy"
   TextField "Text field_9" at 56,281 size 198x18; Text 'Preset-процедура активна'
   Circle "Circle_8" at 28,302 size 16x16
      Appearance <- "PresetDone"
   TextField "Text field_10" at 56,301 size 191x18; Text 'Preset успішно виконано.'
   Circle "Circle_15" at 28,322 size 16x16
      Appearance <- "PresetError"
   TextField "Text field_11" at 56,321 size 198x18; Text 'Помилка виконання preset'
   TextField "Text field_13" at 414,249 size 127x18; Text 'Статус енкодеру'
   TextField "Text field_21" at 414,221 size 115x18; Text 'Статус пресету'
   SymbolicIOField "Symbolic I/O field_1" at 562,214 size 230x32; TextOff '0'; TextOn '1'; TextList "PresetStatus"
      ProcessValue <- "PresetStatus"
   SymbolicIOField "Symbolic I/O field_2" at 562,242 size 230x32; TextOff '0'; TextOn '1'; TextList "EncoderStatus"
      ProcessValue <- "Status"
   TextField "Text field_22" at 308,6 size 185x23; Text 'Стан енкодеру 1BR'

screen "41_РегістраціяПодій" 800x454, template "Template_1"
   on GenerateScreen: SetTag("Tag_ScreenNumber", 41); SetTag("iVisibilityDevices", 0)
   AlarmView "alwContactor" at 119,29 size 675x370; ColumnTextDate 'Дата'; ColumnTextTime 'Час'; ColumnTextAlarmText 'Повідомлення'; ColumnTextAlarmState 'Обладнання'; AlarmLog "MessageContactor"
      Visibility <- "iVisibilityDevices"
   AlarmView "alwLiftUp" at 119,29 size 675x370; ColumnTextDate 'Дата'; ColumnTextTime 'Час'; ColumnTextAlarmText 'Повідомлення'; ColumnTextAlarmState 'Обладнання'; AlarmLog "MessageLiftUp"
      Visibility <- "iVisibilityDevices"
   AlarmView "alwTrolley" at 119,29 size 675x370; ColumnTextDate 'Дата'; ColumnTextTime 'Час'; ColumnTextAlarmText 'Повідомлення'; ColumnTextAlarmState 'Обладнання'; AlarmLog "MessageTrolley"
      Visibility <- "iVisibilityDevices"
   AlarmView "alwCrane" at 119,29 size 675x370; ColumnTextDate 'Дата'; ColumnTextTime 'Час'; ColumnTextAlarmText 'Повідомлення'; ColumnTextAlarmState 'Обладнання'; AlarmLog "MessageCrane"
      Visibility <- "iVisibilityDevices"
   AlarmView "alwDiag" at 119,29 size 675x370; ColumnTextDate 'Дата'; ColumnTextTime 'Час'; ColumnTextAlarmText 'Повідомлення'; ColumnTextAlarmState 'Обладнання'; AlarmLog "MessageDiag"
      Visibility <- "iVisibilityDevices"
   Button "btnLiftUp" at 8,120 size 96x32; TextOff 'Механізм підйому'
      on Release: SetTag("iVisibilityDevices", 1)
      Appearance <- "iVisibilityDevices"
   Button "btnTrolley" at 8,160 size 96x32; TextOff 'Механізм візка'
      on Click: SetTag("iVisibilityDevices", 2)
      Appearance <- "iVisibilityDevices"
   Button "btnCrane" at 8,200 size 96x32; TextOff 'Механізм крану'
      on Release: SetTag("iVisibilityDevices", 3)
      Appearance <- "iVisibilityDevices"
   Button "btnContactor" at 8,80 size 96x32; TextOff 'Лінійний контактор'
      on Release: SetTag("iVisibilityDevices", 0)
      Appearance <- "iVisibilityDevices"
   Button "btnCrane_1" at 8,240 size 96x32; TextOff 'Діагностика'
      on Release: SetTag("iVisibilityDevices", 4)
      Appearance <- "iVisibilityDevices"
   Button "Button_1" at 8,367 size 96x32; TextOff 'Аварія'; TextOn 'Діагностика'
      on Release: ActivateScreen("40_Аварії", 0)
   TextField "Text field_1" at 372,5 size 170x23; Text 'Регістрація подій'
   Button "btnSelf" at 8,280 size 96x32; TextOff 'Власні потреби'
      on Release: SetTag("iVisibilityDevices", 5)
      Appearance <- "iVisibilityDevices"
   AlarmView "alwSelf" at 119,29 size 675x370; ColumnTextDate 'Дата'; ColumnTextTime 'Час'; ColumnTextAlarmText 'Повідомлення'; ColumnTextAlarmState 'Обладнання'; AlarmLog "MessageSelf"
      Visibility <- "iVisibilityDevices"

screen "51_Trends(3UZ1)" 800x454, template "Template_1"
   on GenerateScreen: SetTag("iVisibilityDevices", 0); SetTag("Tag_ScreenNumber", 51)
   TrendView "trvCurrent" at 155,10 size 640x200
      Visibility <- "iVisibilityDevices"
   TrendView "trvMoment" at 155,208 size 640x200
      Visibility <- "iVisibilityDevices"
   TextField "txtCurrent" at 125,95 size 19x30; Text 'I ,А'
      Visibility <- "iVisibilityDevices"
   TextField "txtMoment" at 125,278 size 19x60; Text 'M , Н*м'
      Visibility <- "iVisibilityDevices"
   Button "btnLiftUp" at 8,120 size 96x32; TextOff '3UZ1'
   Button "btnTrolley" at 8,160 size 96x32; TextOff '4UZ1'
      on Release: ActivateScreen("52_Trends(4UZ1)", 0)
   Button "btnCrane" at 8,200 size 96x32; TextOff '4UZ2'
      on Release: ActivateScreen("53_Trends(4UZ2)", 0)
   Button "btnContactor" at 8,80 size 96x32; TextOff '1UZ1'
      on Release: ActivateScreen("50_Trends(1UZ1)", 0)
   Button "Button_1" at 8,319 size 96x32; TextOff 'Струм Момент'
      on Release: SetTag("iVisibilityDevices", 0)
      Appearance <- "iVisibilityDevices"
   Button "Button_2" at 8,356 size 96x32; TextOff 'Швидкості'
      on Release: SetTag("iVisibilityDevices", 1)
      Appearance <- "iVisibilityDevices"
   Button "Button_3" at 4,10 size 104x34; TextOff 'Діагностика / Діагностіка'; TextOn 'Діагностика'
      on Release: ActivateScreen("70_Діагностика", 0)
   TrendView "trvSpeed" at 155,10 size 640x200
      Visibility <- "iVisibilityDevices"
   TrendView "trvError" at 155,208 size 640x200
      Visibility <- "iVisibilityDevices"
   TextField "txtSpeed" at 108,84 size 19x53; Text 'W_set,'
      Visibility <- "iVisibilityDevices"
   TextField "txtError" at 125,259 size 19x98; Text 'W_err ,об/хв'
      Visibility <- "iVisibilityDevices"
   TextField "txtSpeed_1" at 120,82 size 19x57; Text 'W_real,'
      Visibility <- "iVisibilityDevices"
   TextField "txtSpeed_2" at 132,87 size 19x46; Text 'об/хв'
      Visibility <- "iVisibilityDevices"

screen "52_Trends(4UZ1)" 800x454, template "Template_1"
   on GenerateScreen: SetTag("iVisibilityDevices", 0); SetTag("Tag_ScreenNumber", 52)
   TrendView "trvCurrent" at 155,10 size 640x200
      Visibility <- "iVisibilityDevices"
   TrendView "trvMoment" at 155,208 size 640x200
      Visibility <- "iVisibilityDevices"
   TextField "txtCurrent" at 125,95 size 19x30; Text 'I ,А'
      Visibility <- "iVisibilityDevices"
   TextField "txtMoment" at 125,278 size 19x60; Text 'M , Н*м'
      Visibility <- "iVisibilityDevices"
   Button "btnLiftUp" at 8,120 size 96x32; TextOff '3UZ1'
      on Release: ActivateScreen("51_Trends(3UZ1)", 0)
   Button "btnTrolley" at 8,160 size 96x32; TextOff '4UZ1'
   Button "btnCrane" at 8,200 size 96x32; TextOff '4UZ2'
      on Release: ActivateScreen("53_Trends(4UZ2)", 0)
   Button "btnContactor" at 8,80 size 96x32; TextOff '1UZ1'
      on Release: ActivateScreen("50_Trends(1UZ1)", 0)
   Button "Button_1" at 8,319 size 96x32; TextOff 'Струм Момент'
      on Release: SetTag("iVisibilityDevices", 0)
      Appearance <- "iVisibilityDevices"
   Button "Button_2" at 8,356 size 96x32; TextOff 'Швидкості'
      on Release: SetTag("iVisibilityDevices", 1)
      Appearance <- "iVisibilityDevices"
   Button "Button_3" at 4,10 size 104x34; TextOff 'Діагностика / Діагностіка'; TextOn 'Діагностика'
      on Release: ActivateScreen("70_Діагностика", 0)
   TrendView "trvSpeed" at 155,10 size 640x200
      Visibility <- "iVisibilityDevices"
   TrendView "trvError" at 155,208 size 640x200
      Visibility <- "iVisibilityDevices"
   TextField "txtSpeed" at 108,84 size 19x53; Text 'W_set,'
      Visibility <- "iVisibilityDevices"
   TextField "txtError" at 125,259 size 19x98; Text 'W_err ,об/хв'
      Visibility <- "iVisibilityDevices"
   TextField "txtSpeed_1" at 120,82 size 19x57; Text 'W_real,'
      Visibility <- "iVisibilityDevices"
   TextField "txtSpeed_2" at 132,87 size 19x46; Text 'об/хв'
      Visibility <- "iVisibilityDevices"

screen "53_Trends(4UZ2)" 800x454, template "Template_1"
   on GenerateScreen: SetTag("iVisibilityDevices", 0); SetTag("Tag_ScreenNumber", 53)
   TrendView "trvCurrent" at 155,10 size 640x200
      Visibility <- "iVisibilityDevices"
   TrendView "trvMoment" at 155,208 size 640x200
      Visibility <- "iVisibilityDevices"
   TextField "txtCurrent" at 125,95 size 19x30; Text 'I ,А'
      Visibility <- "iVisibilityDevices"
   TextField "txtMoment" at 125,278 size 19x60; Text 'M , Н*м'
      Visibility <- "iVisibilityDevices"
   Button "btnLiftUp" at 8,120 size 96x32; TextOff '3UZ1'
      on Release: ActivateScreen("51_Trends(3UZ1)", 0)
   Button "btnTrolley" at 8,160 size 96x32; TextOff '4UZ1'
      on Release: ActivateScreen("52_Trends(4UZ1)", 0)
   Button "btnCrane" at 8,200 size 96x32; TextOff '4UZ2'
   Button "btnContactor" at 8,80 size 96x32; TextOff '1UZ1'
      on Release: ActivateScreen("50_Trends(1UZ1)", 0)
   Button "Button_1" at 8,319 size 96x32; TextOff 'Струм Момент'
      on Release: SetTag("iVisibilityDevices", 0)
      Appearance <- "iVisibilityDevices"
   Button "Button_2" at 8,356 size 96x32; TextOff 'Швидкості'
      on Release: SetTag("iVisibilityDevices", 1)
      Appearance <- "iVisibilityDevices"
   Button "Button_3" at 4,10 size 104x34; TextOff 'Діагностика / Діагностіка'; TextOn 'Діагностика'
      on Release: ActivateScreen("70_Діагностика", 0)
   TrendView "trvSpeed" at 155,10 size 640x200
      Visibility <- "iVisibilityDevices"
   TrendView "trvError" at 155,208 size 640x200
      Visibility <- "iVisibilityDevices"
   TextField "txtSpeed" at 108,84 size 19x53; Text 'W_set,'
      Visibility <- "iVisibilityDevices"
   TextField "txtError" at 125,259 size 19x98; Text 'W_err ,об/хв'
      Visibility <- "iVisibilityDevices"
   TextField "txtSpeed_1" at 120,82 size 19x57; Text 'W_real,'
      Visibility <- "iVisibilityDevices"
   TextField "txtSpeed_2" at 132,87 size 19x46; Text 'об/хв'
      Visibility <- "iVisibilityDevices"

screen "31_Drives(1UZ1)" 800x454, template "Template_1"
   on GenerateScreen: SetTag("Tag_ScreenNumber", 31); SetTag("iVisibilityDevices", 0)
   Rectangle "rctCU320" at 7,79 size 98x34
      Visibility <- "Error"
   Rectangle "rct1UZ1" at 7,119 size 98x34
      Visibility <- "Error"
   Rectangle "rct4UZ1" at 7,199 size 98x34
      Visibility <- "Error"
   Rectangle "rct3UZ1" at 7,159 size 98x34
      Visibility <- "Error"
   Button "btn1UZ1" at 8,120 size 96x32; TextOff '1UZ1'
   Button "btn3UZ1" at 8,160 size 96x32; TextOff '3UZ1'
      on Release: ActivateScreen("32_Drives(3UZ1)", 0)
   Button "btn4UZ1" at 8,200 size 96x32; TextOff '4UZ1'
      on Release: ActivateScreen("33_Drives(4UZ1)", 0)
   Button "btnCU320" at 8,80 size 96x32; TextOff 'Модуль Кер. CU320 - 2PN'
      on Release: ActivateScreen("30_Drives(CU)", 0)
   Rectangle "rct4UZ2" at 7,239 size 98x34
      Visibility <- "Error"
   Button "btn4UZ2" at 8,240 size 96x32; TextOff '4UZ2'
      on Release: ActivateScreen("34_Drives(4UZ2)", 0)
   Button "Button_1" at 8,319 size 96x32; TextOff 'Телеграмма'
      on Release: SetTag("iVisibilityDevices", 0)
      Appearance <- "iVisibilityDevices"
   Button "Button_2" at 8,356 size 96x32; TextOff 'Значення'
      on Release: SetTag("iVisibilityDevices", 1)
      Appearance <- "iVisibilityDevices"
   Circle "Circle_12" at 130,54 size 16x16
      Visibility <- "iVisibilityDevices"
      Appearance <- "OnOff1"
   TextField "Text field_15" at 158,53 size 250x18; Text 'ON / OFF1'
      Visibility <- "iVisibilityDevices"
   Circle "Circle_13" at 130,74 size 16x16
      Visibility <- "iVisibilityDevices"
      Appearance <- "NoCoastStop"
   TextField "Text field_16" at 158,73 size 250x18; Text 'OFF2 не активний'
      Visibility <- "iVisibilityDevices"
   Circle "Circle_14" at 441,54 size 16x16
      Visibility <- "iVisibilityDevices"
      Appearance <- "ReadyToSwitchOn"
   TextField "Text field_17" at 469,53 size 250x18; Text 'ПЧ готовий до вмикання'
      Visibility <- "iVisibilityDevices"
   Circle "Circle_15" at 441,74 size 16x16
      Visibility <- "iVisibilityDevices"
      Appearance <- "ReadyToOperate"
   TextField "Text field_18" at 469,73 size 250x18; Text 'ПЧ готовий до роботи'
      Visibility <- "iVisibilityDevices"
   Circle "Circle_16" at 441,94 size 16x16
      Visibility <- "iVisibilityDevices"
      Appearance <- "OperationEnabled"
   TextField "Text field_19" at 469,93 size 250x18; Text 'Робота дозволена / стан ОК'
      Visibility <- "iVisibilityDevices"
   Circle "Circle_17" at 441,114 size 16x16
      Visibility <- "iVisibilityDevices"
      Appearance <- "FaultActive"
   TextField "Text field_20" at 469,113 size 250x18; Text 'Аварія ПЧ'
      Visibility <- "iVisibilityDevices"
   Circle "Circle_18" at 441,134 size 16x16
      Visibility <- "iVisibilityDevices"
      Appearance <- "NoCoastStopActive"
   TextField "Text field_21" at 469,133 size 250x18; Text 'OFF2 не активний'
      Visibility <- "iVisibilityDevices"
   Circle "Circle_19" at 441,154 size 16x16
      Visibility <- "iVisibilityDevices"
      Appearance <- "NoQuickStopActive"
   TextField "Text field_22" at 469,153 size 250x18; Text 'OFF3 / Quick Stop не активний'
      Visibility <- "iVisibilityDevices"
   Circle "Circle_20" at 441,174 size 16x16
      Visibility <- "iVisibilityDevices"
      Appearance <- "SwitchingOnInhibit"
   TextField "Text field_23" at 469,173 size 250x18; Text 'Заборона вмикання / блокування'
      Visibility <- "iVisibilityDevices"
   Circle "Circle_21" at 441,194 size 16x16
      Visibility <- "iVisibilityDevices"
      Appearance <- "WarningActive"
   TextField "Text field_24" at 469,193 size 250x18; Text 'Попередження ПЧ'
      Visibility <- "iVisibilityDevices"
   Circle "Circle_22" at 441,214 size 16x16
      Visibility <- "iVisibilityDevices"
      Appearance <- "SpeedErrorInTolerance"
   TextField "Text field_25" at 469,213 size 250x18; Text 'Відхилення швидкості у межах'
      Visibility <- "iVisibilityDevices"
   TextField "Text field_26" at 119,23 size 154x21; Text 'Слово керування:'
      Visibility <- "iVisibilityDevices"
   TextField "Text field_27" at 430,23 size 127x21; Text 'Слово статусу:'
      Visibility <- "iVisibilityDevices"
   Circle "Circle_23" at 130,94 size 16x16
      Visibility <- "iVisibilityDevices"
      Appearance <- "NoQuickStop"
   TextField "Text field_29" at 158,93 size 250x18; Text 'OFF3 / Quick Stop не актвивний'
      Visibility <- "iVisibilityDevices"
   Circle "Circle_24" at 130,114 size 16x16
      Visibility <- "iVisibilityDevices"
      Appearance <- "EnableOperation"
   TextField "Text field_30" at 158,113 size 250x18; Text 'Дозвіл роботи ПЧ'
      Visibility <- "iVisibilityDevices"
   Circle "Circle_25" at 130,134 size 16x16
      Visibility <- "iVisibilityDevices"
      Appearance <- "RampGeneratorEnable"
   TextField "Text field_31" at 158,133 size 250x18; Text 'Дозвіл генератора рампи'
      Visibility <- "iVisibilityDevices"
   Circle "Circle_26" at 130,154 size 16x16
      Visibility <- "iVisibilityDevices"
      Appearance <- "RampGeneratorContinue"
   TextField "Text field_32" at 158,153 size 270x18; Text 'Продовження роботи генератора рампи'
      Visibility <- "iVisibilityDevices"
   Circle "Circle_27" at 130,174 size 16x16
      Visibility <- "iVisibilityDevices"
      Appearance <- "SetpointEnable"
   TextField "Text field_33" at 158,173 size 250x18; Text 'Дозвіл завданяя швидкості'
      Visibility <- "iVisibilityDevices"
   Circle "Circle_28" at 130,194 size 16x16
      Visibility <- "iVisibilityDevices"
      Appearance <- "FaultAcknowledge"
   TextField "Text field_34" at 158,193 size 250x18; Text 'Квітування аварії ПЧ'
      Visibility <- "iVisibilityDevices"
   Circle "Circle_29" at 130,214 size 16x16
      Visibility <- "iVisibilityDevices"
      Appearance <- "ControlByPLC"
   TextField "Text field_35" at 158,213 size 250x18; Text 'Керування від PLC'
      Visibility <- "iVisibilityDevices"
   Circle "Circle_30" at 441,234 size 16x16
      Visibility <- "iVisibilityDevices"
      Appearance <- "ControlRequested"
   TextField "Text field_36" at 469,233 size 250x18; Text 'Керування від PLC'
      Visibility <- "iVisibilityDevices"
   Circle "Circle_31" at 441,254 size 16x16
      Visibility <- "iVisibilityDevices"
      Appearance <- "SetpointReached"
   TextField "Text field_37" at 469,253 size 250x18; Text 'Завдання досягнуто'
      Visibility <- "iVisibilityDevices"
   Circle "Circle_32" at 441,274 size 16x16
      Visibility <- "iVisibilityDevices"
      Appearance <- "InternalLimitActive"
   TextField "Text field_38" at 469,273 size 250x18; Text 'Внутрішнє обмеження'
      Visibility <- "iVisibilityDevices"
   TextField "Text field_39" at 119,338 size 164x21; Text 'Попередження ПЧ:'
      Visibility <- "iVisibilityDevices"
   TextField "Text field_40" at 119,364 size 93x21; Text 'Аварія ПЧ:'
      Visibility <- "iVisibilityDevices"
   SymbolicIOField "Symbolic I/O field_3" at 294,333 size 480x32; TextOff '0'; TextOn '1'; TextList "WarningList"
      ProcessValue <- "WarningCode"
      Visibility <- "iVisibilityDevices"
   SymbolicIOField "Symbolic I/O field_4" at 294,359 size 480x32; TextOff '0'; TextOn '1'; TextList "AlarmList"
      ProcessValue <- "FaultCode"
      Visibility <- "iVisibilityDevices"
   TextField "Text field_7" at 441,304 size 164x18; Text 'Факт. швидк, об / хв:'
      Visibility <- "iVisibilityDevices"
   TextField "Text field_8" at 130,244 size 163x18; Text 'Завд. швидк, об / хв:'
      Visibility <- "iVisibilityDevices"
   IOField "I/O field_7" at 619,297 size 120x32; FormatPattern s9999.99; Unit  об/хв
      ProcessValue <- "ActVelocity_Rpm"
      Visibility <- "iVisibilityDevices"
   IOField "I/O field_8" at 308,237 size 120x32; FormatPattern s9999.99; Unit  об/хв
      ProcessValue <- "SpeedSetpointFb_Rpm"
      Visibility <- "iVisibilityDevices"
   TextField "Text field_1" at 130,54 size 219x18; Text 'Фактична швидкість, об / хв:'
      Visibility <- "iVisibilityDevices"
   TextField "Text field_2" at 130,77 size 220x18; Text 'Завдання швидкості, об / хв:'
      Visibility <- "iVisibilityDevices"
   TextField "Text field_3" at 130,100 size 74x18; Text 'Струм, А:'
      Visibility <- "iVisibilityDevices"
   TextField "Text field_4" at 130,123 size 105x18; Text 'Момент, Н*м:'
      Visibility <- "iVisibilityDevices"
   TextField "Text field_5" at 130,146 size 128x18; Text 'Потужність, кВТ:'
      Visibility <- "iVisibilityDevices"
   TextField "Text field_6" at 130,169 size 139x18; Text 'Завантаження, %:'
      Visibility <- "iVisibilityDevices"
   IOField "I/O field_1" at 376,47 size 120x32; FormatPattern s9999.99; Unit  об/хв
      ProcessValue <- "ActVelocity_Rpm"
      Visibility <- "iVisibilityDevices"
   IOField "I/O field_2" at 376,70 size 120x32; FormatPattern s9999.99; Unit  об/хв
      ProcessValue <- "SpeedSetpointFb_Rpm"
      Visibility <- "iVisibilityDevices"
   IOField "I/O field_3" at 376,93 size 120x32; FormatPattern s9999.99; Unit  А
      ProcessValue <- "ActCurrent_A"
      Visibility <- "iVisibilityDevices"
   IOField "I/O field_4" at 376,116 size 120x32; FormatPattern s9999.99; Unit  Н*м
      ProcessValue <- "ActTorque_Nm"
      Visibility <- "iVisibilityDevices"
   IOField "I/O field_5" at 376,139 size 120x32; FormatPattern s9999.99; Unit  кВт
      ProcessValue <- "ActPower_kW"
      Visibility <- "iVisibilityDevices"
   IOField "I/O field_6" at 376,162 size 120x32; FormatPattern s9999.99; Unit  %
      ProcessValue <- "LoadPower_Pct"
      Visibility <- "iVisibilityDevices"

screen "32_Drives(3UZ1)" 800x454, template "Template_1"
   on GenerateScreen: SetTag("Tag_ScreenNumber", 32); SetTag("iVisibilityDevices", 0)
   Rectangle "rctCU320" at 7,79 size 98x34
      Visibility <- "Error"
   Rectangle "rct1UZ1" at 7,119 size 98x34
      Visibility <- "Error"
   Rectangle "rct4UZ1" at 7,199 size 98x34
      Visibility <- "Error"
   Rectangle "rct3UZ1" at 7,159 size 98x34
      Visibility <- "Error"
   Button "btn1UZ1" at 8,120 size 96x32; TextOff '1UZ1'
      on Release: ActivateScreen("31_Drives(1UZ1)", 0)
   Button "btn3UZ1" at 8,160 size 96x32; TextOff '3UZ1'
   Button "btn4UZ1" at 8,200 size 96x32; TextOff '4UZ1'
      on Release: ActivateScreen("33_Drives(4UZ1)", 0)
   Button "btnCU320" at 8,80 size 96x32; TextOff 'Модуль Кер. CU320 - 2PN'
      on Release: ActivateScreen("30_Drives(CU)", 0)
   Rectangle "rct4UZ2" at 7,239 size 98x34
      Visibility <- "Error"
   Button "btn4UZ2" at 8,240 size 96x32; TextOff '4UZ2'
      on Release: ActivateScreen("34_Drives(4UZ2)", 0)
   Button "Button_1" at 8,319 size 96x32; TextOff 'Телеграмма'
      on Release: SetTag("iVisibilityDevices", 0)
      Appearance <- "iVisibilityDevices"
   Button "Button_2" at 8,356 size 96x32; TextOff 'Значення'
      on Release: SetTag("iVisibilityDevices", 1)
      Appearance <- "iVisibilityDevices"
   Circle "Circle_12" at 130,54 size 16x16
      Visibility <- "iVisibilityDevices"
      Appearance <- "OnOff1"
   TextField "Text field_15" at 158,53 size 250x18; Text 'ON / OFF1'
      Visibility <- "iVisibilityDevices"
   Circle "Circle_13" at 130,74 size 16x16
      Visibility <- "iVisibilityDevices"
      Appearance <- "NoCoastStop"
   TextField "Text field_16" at 158,73 size 250x18; Text 'OFF2 не активний'
      Visibility <- "iVisibilityDevices"
   Circle "Circle_14" at 441,54 size 16x16
      Visibility <- "iVisibilityDevices"
      Appearance <- "ReadyToSwitchOn"
   TextField "Text field_17" at 469,53 size 250x18; Text 'ПЧ готовий до вмикання'
      Visibility <- "iVisibilityDevices"
   Circle "Circle_15" at 441,74 size 16x16
      Visibility <- "iVisibilityDevices"
      Appearance <- "ReadyToOperate"
   TextField "Text field_18" at 469,73 size 250x18; Text 'ПЧ готовий до роботи'
      Visibility <- "iVisibilityDevices"
   Circle "Circle_16" at 441,94 size 16x16
      Visibility <- "iVisibilityDevices"
      Appearance <- "OperationEnabled"
   TextField "Text field_19" at 469,93 size 250x18; Text 'Робота дозволена / стан ОК'
      Visibility <- "iVisibilityDevices"
   Circle "Circle_17" at 441,114 size 16x16
      Visibility <- "iVisibilityDevices"
      Appearance <- "FaultActive"
   TextField "Text field_20" at 469,113 size 250x18; Text 'Аварія ПЧ'
      Visibility <- "iVisibilityDevices"
   Circle "Circle_18" at 441,134 size 16x16
      Visibility <- "iVisibilityDevices"
      Appearance <- "NoCoastStopActive"
   TextField "Text field_21" at 469,133 size 250x18; Text 'OFF2 не активний'
      Visibility <- "iVisibilityDevices"
   Circle "Circle_19" at 441,154 size 16x16
      Visibility <- "iVisibilityDevices"
      Appearance <- "NoQuickStopActive"
   TextField "Text field_22" at 469,153 size 250x18; Text 'OFF3 / Quick Stop не активний'
      Visibility <- "iVisibilityDevices"
   Circle "Circle_20" at 441,174 size 16x16
      Visibility <- "iVisibilityDevices"
      Appearance <- "SwitchingOnInhibit"
   TextField "Text field_23" at 469,173 size 250x18; Text 'Заборона вмикання / блокування'
      Visibility <- "iVisibilityDevices"
   Circle "Circle_21" at 441,194 size 16x16
      Visibility <- "iVisibilityDevices"
      Appearance <- "WarningActive"
   TextField "Text field_24" at 469,193 size 250x18; Text 'Попередження ПЧ'
      Visibility <- "iVisibilityDevices"
   Circle "Circle_22" at 441,214 size 16x16
      Visibility <- "iVisibilityDevices"
      Appearance <- "SpeedErrorInTolerance"
   TextField "Text field_25" at 469,213 size 250x18; Text 'Відхилення швидкості у межах'
      Visibility <- "iVisibilityDevices"
   TextField "Text field_26" at 119,23 size 154x21; Text 'Слово керування:'
      Visibility <- "iVisibilityDevices"
   TextField "Text field_27" at 430,23 size 127x21; Text 'Слово статусу:'
      Visibility <- "iVisibilityDevices"
   Circle "Circle_23" at 130,94 size 16x16
      Visibility <- "iVisibilityDevices"
      Appearance <- "NoQuickStop"
   TextField "Text field_29" at 158,93 size 250x18; Text 'OFF3 / Quick Stop не актвивний'
      Visibility <- "iVisibilityDevices"
   Circle "Circle_24" at 130,114 size 16x16
      Visibility <- "iVisibilityDevices"
      Appearance <- "EnableOperation"
   TextField "Text field_30" at 158,113 size 250x18; Text 'Дозвіл роботи ПЧ'
      Visibility <- "iVisibilityDevices"
   Circle "Circle_25" at 130,134 size 16x16
      Visibility <- "iVisibilityDevices"
      Appearance <- "RampGeneratorEnable"
   TextField "Text field_31" at 158,133 size 250x18; Text 'Дозвіл генератора рампи'
      Visibility <- "iVisibilityDevices"
   Circle "Circle_26" at 130,154 size 16x16
      Visibility <- "iVisibilityDevices"
      Appearance <- "RampGeneratorContinue"
   TextField "Text field_32" at 158,153 size 270x18; Text 'Продовження роботи генератора рампи'
      Visibility <- "iVisibilityDevices"
   Circle "Circle_27" at 130,174 size 16x16
      Visibility <- "iVisibilityDevices"
      Appearance <- "SetpointEnable"
   TextField "Text field_33" at 158,173 size 250x18; Text 'Дозвіл завданяя швидкості'
      Visibility <- "iVisibilityDevices"
   Circle "Circle_28" at 130,194 size 16x16
      Visibility <- "iVisibilityDevices"
      Appearance <- "FaultAcknowledge"
   TextField "Text field_34" at 158,193 size 250x18; Text 'Квітування аварії ПЧ'
      Visibility <- "iVisibilityDevices"
   Circle "Circle_29" at 130,214 size 16x16
      Visibility <- "iVisibilityDevices"
      Appearance <- "ControlByPLC"
   TextField "Text field_35" at 158,213 size 250x18; Text 'Керування від PLC'
      Visibility <- "iVisibilityDevices"
   Circle "Circle_30" at 441,234 size 16x16
      Visibility <- "iVisibilityDevices"
      Appearance <- "ControlRequested"
   TextField "Text field_36" at 469,233 size 250x18; Text 'Керування від PLC'
      Visibility <- "iVisibilityDevices"
   Circle "Circle_31" at 441,254 size 16x16
      Visibility <- "iVisibilityDevices"
      Appearance <- "SetpointReached"
   TextField "Text field_37" at 469,253 size 250x18; Text 'Завдання досягнуто'
      Visibility <- "iVisibilityDevices"
   Circle "Circle_32" at 441,274 size 16x16
      Visibility <- "iVisibilityDevices"
      Appearance <- "InternalLimitActive"
   TextField "Text field_38" at 469,273 size 250x18; Text 'Внутрішнє обмеження'
      Visibility <- "iVisibilityDevices"
   TextField "Text field_39" at 119,338 size 164x21; Text 'Попередження ПЧ:'
      Visibility <- "iVisibilityDevices"
   TextField "Text field_40" at 119,364 size 93x21; Text 'Аварія ПЧ:'
      Visibility <- "iVisibilityDevices"
   SymbolicIOField "Symbolic I/O field_3" at 294,333 size 480x32; TextOff '0'; TextOn '1'; TextList "WarningList"
      Visibility <- "iVisibilityDevices"
      ProcessValue <- "WarningCode"
   SymbolicIOField "Symbolic I/O field_4" at 294,359 size 480x32; TextOff '0'; TextOn '1'; TextList "AlarmList"
      Visibility <- "iVisibilityDevices"
      ProcessValue <- "FaultCode"
   TextField "Text field_7" at 441,304 size 164x18; Text 'Факт. швидк, об / хв:'
      Visibility <- "iVisibilityDevices"
   TextField "Text field_8" at 130,244 size 163x18; Text 'Завд. швидк, об / хв:'
      Visibility <- "iVisibilityDevices"
   IOField "I/O field_7" at 619,297 size 120x32; FormatPattern s9999.99; Unit  об/хв
      Visibility <- "iVisibilityDevices"
      ProcessValue <- "ActVelocity_Rpm"
   IOField "I/O field_8" at 308,237 size 120x32; FormatPattern s9999.99; Unit  об/хв
      Visibility <- "iVisibilityDevices"
      ProcessValue <- "SpeedSetpointFb_Rpm"
   TextField "Text field_1" at 130,54 size 219x18; Text 'Фактична швидкість, об / хв:'
      Visibility <- "iVisibilityDevices"
   TextField "Text field_2" at 130,77 size 220x18; Text 'Завдання швидкості, об / хв:'
      Visibility <- "iVisibilityDevices"
   TextField "Text field_3" at 130,100 size 74x18; Text 'Струм, А:'
      Visibility <- "iVisibilityDevices"
   TextField "Text field_4" at 130,123 size 105x18; Text 'Момент, Н*м:'
      Visibility <- "iVisibilityDevices"
   TextField "Text field_5" at 130,146 size 128x18; Text 'Потужність, кВТ:'
      Visibility <- "iVisibilityDevices"
   TextField "Text field_6" at 130,169 size 139x18; Text 'Завантаження, %:'
      Visibility <- "iVisibilityDevices"
   IOField "I/O field_1" at 376,47 size 120x32; FormatPattern s9999.99; Unit  об/хв
      Visibility <- "iVisibilityDevices"
      ProcessValue <- "ActVelocity_Rpm"
   IOField "I/O field_2" at 376,70 size 120x32; FormatPattern s9999.99; Unit  об/хв
      Visibility <- "iVisibilityDevices"
      ProcessValue <- "SpeedSetpointFb_Rpm"
   IOField "I/O field_3" at 376,93 size 120x32; FormatPattern s9999.99; Unit  А
      Visibility <- "iVisibilityDevices"
      ProcessValue <- "ActCurrent_A"
   IOField "I/O field_4" at 376,116 size 120x32; FormatPattern s9999.99; Unit  Н*м
      Visibility <- "iVisibilityDevices"
      ProcessValue <- "ActTorque_Nm"
   IOField "I/O field_5" at 376,139 size 120x32; FormatPattern s9999.99; Unit  кВт
      Visibility <- "iVisibilityDevices"
      ProcessValue <- "ActPower_kW"
   IOField "I/O field_6" at 376,162 size 120x32; FormatPattern s9999.99; Unit  %
      Visibility <- "iVisibilityDevices"
      ProcessValue <- "LoadPower_Pct"

screen "33_Drives(4UZ1)" 800x454, template "Template_1"
   on GenerateScreen: SetTag("Tag_ScreenNumber", 33); SetTag("iVisibilityDevices", 0)
   Rectangle "rctCU320" at 7,79 size 98x34
      Visibility <- "Error"
   Rectangle "rct1UZ1" at 7,119 size 98x34
      Visibility <- "Error"
   Rectangle "rct4UZ1" at 7,199 size 98x34
      Visibility <- "Error"
   Rectangle "rct3UZ1" at 7,159 size 98x34
      Visibility <- "Error"
   Button "btn1UZ1" at 8,120 size 96x32; TextOff '1UZ1'
      on Release: ActivateScreen("31_Drives(1UZ1)", 0)
   Button "btn3UZ1" at 8,160 size 96x32; TextOff '3UZ1'
      on Release: ActivateScreen("32_Drives(3UZ1)", 0)
   Button "btn4UZ1" at 8,200 size 96x32; TextOff '4UZ1'
   Button "btnCU320" at 8,80 size 96x32; TextOff 'Модуль Кер. CU320 - 2PN'
      on Release: ActivateScreen("30_Drives(CU)", 0)
   Rectangle "rct4UZ2" at 7,239 size 98x34
      Visibility <- "Error"
   Button "btn4UZ2" at 8,240 size 96x32; TextOff '4UZ2'
      on Release: ActivateScreen("34_Drives(4UZ2)", 0)
   Button "Button_1" at 8,319 size 96x32; TextOff 'Телеграмма'
      on Release: SetTag("iVisibilityDevices", 0)
      Appearance <- "iVisibilityDevices"
   Button "Button_2" at 8,356 size 96x32; TextOff 'Значення'
      on Release: SetTag("iVisibilityDevices", 1)
      Appearance <- "iVisibilityDevices"
   Circle "Circle_12" at 130,54 size 16x16
      Visibility <- "iVisibilityDevices"
      Appearance <- "OnOff1"
   TextField "Text field_15" at 158,53 size 250x18; Text 'ON / OFF1'
      Visibility <- "iVisibilityDevices"
   Circle "Circle_13" at 130,74 size 16x16
      Visibility <- "iVisibilityDevices"
      Appearance <- "NoCoastStop"
   TextField "Text field_16" at 158,73 size 250x18; Text 'OFF2 не активний'
      Visibility <- "iVisibilityDevices"
   Circle "Circle_14" at 441,54 size 16x16
      Visibility <- "iVisibilityDevices"
      Appearance <- "ReadyToSwitchOn"
   TextField "Text field_17" at 469,53 size 250x18; Text 'ПЧ готовий до вмикання'
      Visibility <- "iVisibilityDevices"
   Circle "Circle_15" at 441,74 size 16x16
      Visibility <- "iVisibilityDevices"
      Appearance <- "ReadyToOperate"
   TextField "Text field_18" at 469,73 size 250x18; Text 'ПЧ готовий до роботи'
      Visibility <- "iVisibilityDevices"
   Circle "Circle_16" at 441,94 size 16x16
      Visibility <- "iVisibilityDevices"
      Appearance <- "OperationEnabled"
   TextField "Text field_19" at 469,93 size 250x18; Text 'Робота дозволена / стан ОК'
      Visibility <- "iVisibilityDevices"
   Circle "Circle_17" at 441,114 size 16x16
      Visibility <- "iVisibilityDevices"
      Appearance <- "FaultActive"
   TextField "Text field_20" at 469,113 size 250x18; Text 'Аварія ПЧ'
      Visibility <- "iVisibilityDevices"
   Circle "Circle_18" at 441,134 size 16x16
      Visibility <- "iVisibilityDevices"
      Appearance <- "NoCoastStopActive"
   TextField "Text field_21" at 469,133 size 250x18; Text 'OFF2 не активний'
      Visibility <- "iVisibilityDevices"
   Circle "Circle_19" at 441,154 size 16x16
      Visibility <- "iVisibilityDevices"
      Appearance <- "NoQuickStopActive"
   TextField "Text field_22" at 469,153 size 250x18; Text 'OFF3 / Quick Stop не активний'
      Visibility <- "iVisibilityDevices"
   Circle "Circle_20" at 441,174 size 16x16
      Visibility <- "iVisibilityDevices"
      Appearance <- "SwitchingOnInhibit"
   TextField "Text field_23" at 469,173 size 250x18; Text 'Заборона вмикання / блокування'
      Visibility <- "iVisibilityDevices"
   Circle "Circle_21" at 441,194 size 16x16
      Visibility <- "iVisibilityDevices"
      Appearance <- "WarningActive"
   TextField "Text field_24" at 469,193 size 250x18; Text 'Попередження ПЧ'
      Visibility <- "iVisibilityDevices"
   Circle "Circle_22" at 441,214 size 16x16
      Visibility <- "iVisibilityDevices"
      Appearance <- "SpeedErrorInTolerance"
   TextField "Text field_25" at 469,213 size 250x18; Text 'Відхилення швидкості у межах'
      Visibility <- "iVisibilityDevices"
   TextField "Text field_26" at 119,23 size 154x21; Text 'Слово керування:'
      Visibility <- "iVisibilityDevices"
   TextField "Text field_27" at 430,23 size 127x21; Text 'Слово статусу:'
      Visibility <- "iVisibilityDevices"
   Circle "Circle_23" at 130,94 size 16x16
      Visibility <- "iVisibilityDevices"
      Appearance <- "NoQuickStop"
   TextField "Text field_29" at 158,93 size 250x18; Text 'OFF3 / Quick Stop не актвивний'
      Visibility <- "iVisibilityDevices"
   Circle "Circle_24" at 130,114 size 16x16
      Visibility <- "iVisibilityDevices"
      Appearance <- "EnableOperation"
   TextField "Text field_30" at 158,113 size 250x18; Text 'Дозвіл роботи ПЧ'
      Visibility <- "iVisibilityDevices"
   Circle "Circle_25" at 130,134 size 16x16
      Visibility <- "iVisibilityDevices"
      Appearance <- "RampGeneratorEnable"
   TextField "Text field_31" at 158,133 size 250x18; Text 'Дозвіл генератора рампи'
      Visibility <- "iVisibilityDevices"
   Circle "Circle_26" at 130,154 size 16x16
      Visibility <- "iVisibilityDevices"
      Appearance <- "RampGeneratorContinue"
   TextField "Text field_32" at 158,153 size 270x18; Text 'Продовження роботи генератора рампи'
      Visibility <- "iVisibilityDevices"
   Circle "Circle_27" at 130,174 size 16x16
      Visibility <- "iVisibilityDevices"
      Appearance <- "SetpointEnable"
   TextField "Text field_33" at 158,173 size 250x18; Text 'Дозвіл завданяя швидкості'
      Visibility <- "iVisibilityDevices"
   Circle "Circle_28" at 130,194 size 16x16
      Visibility <- "iVisibilityDevices"
      Appearance <- "FaultAcknowledge"
   TextField "Text field_34" at 158,193 size 250x18; Text 'Квітування аварії ПЧ'
      Visibility <- "iVisibilityDevices"
   Circle "Circle_29" at 130,214 size 16x16
      Visibility <- "iVisibilityDevices"
      Appearance <- "ControlByPLC"
   TextField "Text field_35" at 158,213 size 250x18; Text 'Керування від PLC'
      Visibility <- "iVisibilityDevices"
   Circle "Circle_30" at 441,234 size 16x16
      Visibility <- "iVisibilityDevices"
      Appearance <- "ControlRequested"
   TextField "Text field_36" at 469,233 size 250x18; Text 'Керування від PLC'
      Visibility <- "iVisibilityDevices"
   Circle "Circle_31" at 441,254 size 16x16
      Visibility <- "iVisibilityDevices"
      Appearance <- "SetpointReached"
   TextField "Text field_37" at 469,253 size 250x18; Text 'Завдання досягнуто'
      Visibility <- "iVisibilityDevices"
   Circle "Circle_32" at 441,274 size 16x16
      Visibility <- "iVisibilityDevices"
      Appearance <- "InternalLimitActive"
   TextField "Text field_38" at 469,273 size 250x18; Text 'Внутрішнє обмеження'
      Visibility <- "iVisibilityDevices"
   TextField "Text field_39" at 119,338 size 164x21; Text 'Попередження ПЧ:'
      Visibility <- "iVisibilityDevices"
   TextField "Text field_40" at 119,364 size 93x21; Text 'Аварія ПЧ:'
      Visibility <- "iVisibilityDevices"
   SymbolicIOField "Symbolic I/O field_3" at 294,333 size 480x32; TextOff '0'; TextOn '1'; TextList "WarningList"
      Visibility <- "iVisibilityDevices"
      ProcessValue <- "WarningCode"
   SymbolicIOField "Symbolic I/O field_4" at 294,359 size 480x32; TextOff '0'; TextOn '1'; TextList "AlarmList"
      Visibility <- "iVisibilityDevices"
      ProcessValue <- "FaultCode"
   TextField "Text field_7" at 441,304 size 164x18; Text 'Факт. швидк, об / хв:'
      Visibility <- "iVisibilityDevices"
   TextField "Text field_8" at 130,244 size 163x18; Text 'Завд. швидк, об / хв:'
      Visibility <- "iVisibilityDevices"
   IOField "I/O field_7" at 619,297 size 120x32; FormatPattern s9999.99; Unit  об/хв
      Visibility <- "iVisibilityDevices"
      ProcessValue <- "ActVelocity_Rpm"
   IOField "I/O field_8" at 304,237 size 120x32; FormatPattern s9999.99; Unit  об/хв
      Visibility <- "iVisibilityDevices"
      ProcessValue <- "SpeedSetpointFb_Rpm"
   TextField "Text field_1" at 130,54 size 219x18; Text 'Фактична швидкість, об / хв:'
      Visibility <- "iVisibilityDevices"
   TextField "Text field_2" at 130,77 size 220x18; Text 'Завдання швидкості, об / хв:'
      Visibility <- "iVisibilityDevices"
   TextField "Text field_3" at 130,100 size 74x18; Text 'Струм, А:'
      Visibility <- "iVisibilityDevices"
   TextField "Text field_4" at 130,123 size 105x18; Text 'Момент, Н*м:'
      Visibility <- "iVisibilityDevices"
   TextField "Text field_5" at 130,146 size 128x18; Text 'Потужність, кВТ:'
      Visibility <- "iVisibilityDevices"
   TextField "Text field_6" at 130,169 size 139x18; Text 'Завантаження, %:'
      Visibility <- "iVisibilityDevices"
   IOField "I/O field_1" at 376,47 size 120x32; FormatPattern s9999.99; Unit  об/хв
      Visibility <- "iVisibilityDevices"
      ProcessValue <- "ActVelocity_Rpm"
   IOField "I/O field_2" at 376,70 size 120x32; FormatPattern s9999.99; Unit  об/хв
      Visibility <- "iVisibilityDevices"
      ProcessValue <- "SpeedSetpointFb_Rpm"
   IOField "I/O field_3" at 376,93 size 120x32; FormatPattern s9999.99; Unit  А
      Visibility <- "iVisibilityDevices"
      ProcessValue <- "ActCurrent_A"
   IOField "I/O field_4" at 376,116 size 120x32; FormatPattern s9999.99; Unit  Н*м
      Visibility <- "iVisibilityDevices"
      ProcessValue <- "ActTorque_Nm"
   IOField "I/O field_5" at 376,139 size 120x32; FormatPattern s9999.99; Unit  кВт
      Visibility <- "iVisibilityDevices"
      ProcessValue <- "ActPower_kW"
   IOField "I/O field_6" at 376,162 size 120x32; FormatPattern s9999.99; Unit  %
      Visibility <- "iVisibilityDevices"
      ProcessValue <- "LoadPower_Pct"

screen "34_Drives(4UZ2)" 800x454, template "Template_1"
   on GenerateScreen: SetTag("Tag_ScreenNumber", 34); SetTag("iVisibilityDevices", 0)
   Rectangle "rctCU320" at 7,79 size 98x34
      Visibility <- "Error"
   Rectangle "rct1UZ1" at 7,119 size 98x34
      Visibility <- "Error"
   Rectangle "rct4UZ1" at 7,199 size 98x34
      Visibility <- "Error"
   Rectangle "rct3UZ1" at 7,159 size 98x34
      Visibility <- "Error"
   Button "btn1UZ1" at 8,120 size 96x32; TextOff '1UZ1'
      on Release: ActivateScreen("31_Drives(1UZ1)", 0)
   Button "btn3UZ1" at 8,160 size 96x32; TextOff '3UZ1'
      on Release: ActivateScreen("32_Drives(3UZ1)", 0)
   Button "btn4UZ1" at 8,200 size 96x32; TextOff '4UZ1'
      on Release: ActivateScreen("33_Drives(4UZ1)", 0)
   Button "btnCU320" at 8,80 size 96x32; TextOff 'Модуль Кер. CU320 - 2PN'
      on Release: ActivateScreen("30_Drives(CU)", 0)
   Rectangle "rct4UZ2" at 7,239 size 98x34
      Visibility <- "Error"
   Button "btn4UZ2" at 8,240 size 96x32; TextOff '4UZ2'
   Button "Button_1" at 8,319 size 96x32; TextOff 'Телеграмма'
      on Release: SetTag("iVisibilityDevices", 0)
      Appearance <- "iVisibilityDevices"
   Button "Button_2" at 8,356 size 96x32; TextOff 'Значення'
      on Release: SetTag("iVisibilityDevices", 1)
      Appearance <- "iVisibilityDevices"
   Circle "Circle_12" at 130,54 size 16x16
      Visibility <- "iVisibilityDevices"
      Appearance <- "OnOff1"
   TextField "Text field_15" at 158,53 size 250x18; Text 'ON / OFF1'
      Visibility <- "iVisibilityDevices"
   Circle "Circle_13" at 130,74 size 16x16
      Visibility <- "iVisibilityDevices"
      Appearance <- "NoCoastStop"
   TextField "Text field_16" at 158,73 size 250x18; Text 'OFF2 не активний'
      Visibility <- "iVisibilityDevices"
   Circle "Circle_14" at 441,54 size 16x16
      Visibility <- "iVisibilityDevices"
      Appearance <- "ReadyToSwitchOn"
   TextField "Text field_17" at 469,53 size 250x18; Text 'ПЧ готовий до вмикання'
      Visibility <- "iVisibilityDevices"
   Circle "Circle_15" at 441,74 size 16x16
      Visibility <- "iVisibilityDevices"
      Appearance <- "ReadyToOperate"
   TextField "Text field_18" at 469,73 size 250x18; Text 'ПЧ готовий до роботи'
      Visibility <- "iVisibilityDevices"
   Circle "Circle_16" at 441,94 size 16x16
      Visibility <- "iVisibilityDevices"
      Appearance <- "OperationEnabled"
   TextField "Text field_19" at 469,93 size 250x18; Text 'Робота дозволена / стан ОК'
      Visibility <- "iVisibilityDevices"
   Circle "Circle_17" at 441,114 size 16x16
      Visibility <- "iVisibilityDevices"
      Appearance <- "FaultActive"
   TextField "Text field_20" at 469,113 size 250x18; Text 'Аварія ПЧ'
      Visibility <- "iVisibilityDevices"
   Circle "Circle_18" at 441,134 size 16x16
      Visibility <- "iVisibilityDevices"
      Appearance <- "NoCoastStopActive"
   TextField "Text field_21" at 469,133 size 250x18; Text 'OFF2 не активний'
      Visibility <- "iVisibilityDevices"
   Circle "Circle_19" at 441,154 size 16x16
      Visibility <- "iVisibilityDevices"
      Appearance <- "NoQuickStopActive"
   TextField "Text field_22" at 469,153 size 250x18; Text 'OFF3 / Quick Stop не активний'
      Visibility <- "iVisibilityDevices"
   Circle "Circle_20" at 441,174 size 16x16
      Visibility <- "iVisibilityDevices"
      Appearance <- "SwitchingOnInhibit"
   TextField "Text field_23" at 469,173 size 250x18; Text 'Заборона вмикання / блокування'
      Visibility <- "iVisibilityDevices"
   Circle "Circle_21" at 441,194 size 16x16
      Visibility <- "iVisibilityDevices"
      Appearance <- "WarningActive"
   TextField "Text field_24" at 469,193 size 250x18; Text 'Попередження ПЧ'
      Visibility <- "iVisibilityDevices"
   Circle "Circle_22" at 441,214 size 16x16
      Visibility <- "iVisibilityDevices"
      Appearance <- "SpeedErrorInTolerance"
   TextField "Text field_25" at 469,213 size 250x18; Text 'Відхилення швидкості у межах'
      Visibility <- "iVisibilityDevices"
   TextField "Text field_26" at 119,23 size 154x21; Text 'Слово керування:'
      Visibility <- "iVisibilityDevices"
   TextField "Text field_27" at 430,23 size 127x21; Text 'Слово статусу:'
      Visibility <- "iVisibilityDevices"
   Circle "Circle_23" at 130,94 size 16x16
      Visibility <- "iVisibilityDevices"
      Appearance <- "NoQuickStop"
   TextField "Text field_29" at 158,93 size 250x18; Text 'OFF3 / Quick Stop не актвивний'
      Visibility <- "iVisibilityDevices"
   Circle "Circle_24" at 130,114 size 16x16
      Visibility <- "iVisibilityDevices"
      Appearance <- "EnableOperation"
   TextField "Text field_30" at 158,113 size 250x18; Text 'Дозвіл роботи ПЧ'
      Visibility <- "iVisibilityDevices"
   Circle "Circle_25" at 130,134 size 16x16
      Visibility <- "iVisibilityDevices"
      Appearance <- "RampGeneratorEnable"
   TextField "Text field_31" at 158,133 size 250x18; Text 'Дозвіл генератора рампи'
      Visibility <- "iVisibilityDevices"
   Circle "Circle_26" at 130,154 size 16x16
      Visibility <- "iVisibilityDevices"
      Appearance <- "RampGeneratorContinue"
   TextField "Text field_32" at 158,153 size 270x18; Text 'Продовження роботи генератора рампи'
      Visibility <- "iVisibilityDevices"
   Circle "Circle_27" at 130,174 size 16x16
      Visibility <- "iVisibilityDevices"
      Appearance <- "SetpointEnable"
   TextField "Text field_33" at 158,173 size 250x18; Text 'Дозвіл завданяя швидкості'
      Visibility <- "iVisibilityDevices"
   Circle "Circle_28" at 130,194 size 16x16
      Visibility <- "iVisibilityDevices"
      Appearance <- "FaultAcknowledge"
   TextField "Text field_34" at 158,193 size 250x18; Text 'Квітування аварії ПЧ'
      Visibility <- "iVisibilityDevices"
   Circle "Circle_29" at 130,214 size 16x16
      Visibility <- "iVisibilityDevices"
      Appearance <- "ControlByPLC"
   TextField "Text field_35" at 158,213 size 250x18; Text 'Керування від PLC'
      Visibility <- "iVisibilityDevices"
   Circle "Circle_30" at 441,234 size 16x16
      Visibility <- "iVisibilityDevices"
      Appearance <- "ControlRequested"
   TextField "Text field_36" at 469,233 size 250x18; Text 'Керування від PLC'
      Visibility <- "iVisibilityDevices"
   Circle "Circle_31" at 441,254 size 16x16
      Visibility <- "iVisibilityDevices"
      Appearance <- "SetpointReached"
   TextField "Text field_37" at 469,253 size 250x18; Text 'Завдання досягнуто'
      Visibility <- "iVisibilityDevices"
   Circle "Circle_32" at 441,274 size 16x16
      Visibility <- "iVisibilityDevices"
      Appearance <- "InternalLimitActive"
   TextField "Text field_38" at 469,273 size 250x18; Text 'Внутрішнє обмеження'
      Visibility <- "iVisibilityDevices"
   TextField "Text field_39" at 119,338 size 164x21; Text 'Попередження ПЧ:'
      Visibility <- "iVisibilityDevices"
   TextField "Text field_40" at 119,364 size 93x21; Text 'Аварія ПЧ:'
      Visibility <- "iVisibilityDevices"
   SymbolicIOField "Symbolic I/O field_3" at 294,333 size 480x32; TextOff '0'; TextOn '1'; TextList "WarningList"
      Visibility <- "iVisibilityDevices"
      ProcessValue <- "WarningCode"
   SymbolicIOField "Symbolic I/O field_4" at 294,359 size 480x32; TextOff '0'; TextOn '1'; TextList "AlarmList"
      Visibility <- "iVisibilityDevices"
      ProcessValue <- "FaultCode"
   TextField "Text field_7" at 441,304 size 164x18; Text 'Факт. швидк, об / хв:'
      Visibility <- "iVisibilityDevices"
   IOField "I/O field_8" at 304,237 size 120x32; FormatPattern s9999.99; Unit  об/хв
      Visibility <- "iVisibilityDevices"
      ProcessValue <- "SpeedSetpointFb_Rpm"
   TextField "Text field_8" at 130,244 size 163x18; Text 'Завд. швидк, об / хв:'
      Visibility <- "iVisibilityDevices"
   IOField "I/O field_7" at 619,297 size 120x32; FormatPattern s9999.99; Unit  об/хв
      Visibility <- "iVisibilityDevices"
      ProcessValue <- "ActVelocity_Rpm"
   TextField "Text field_1" at 130,54 size 219x18; Text 'Фактична швидкість, об / хв:'
      Visibility <- "iVisibilityDevices"
   TextField "Text field_2" at 130,77 size 220x18; Text 'Завдання швидкості, об / хв:'
      Visibility <- "iVisibilityDevices"
   TextField "Text field_3" at 130,100 size 74x18; Text 'Струм, А:'
      Visibility <- "iVisibilityDevices"
   TextField "Text field_4" at 130,123 size 105x18; Text 'Момент, Н*м:'
      Visibility <- "iVisibilityDevices"
   TextField "Text field_5" at 130,146 size 128x18; Text 'Потужність, кВТ:'
      Visibility <- "iVisibilityDevices"
   TextField "Text field_6" at 130,169 size 139x18; Text 'Завантаження, %:'
      Visibility <- "iVisibilityDevices"
   IOField "I/O field_1" at 376,47 size 120x32; FormatPattern s9999.99; Unit  об/хв
      Visibility <- "iVisibilityDevices"
      ProcessValue <- "ActVelocity_Rpm"
   IOField "I/O field_2" at 376,70 size 120x32; FormatPattern s9999.99; Unit  об/хв
      Visibility <- "iVisibilityDevices"
      ProcessValue <- "SpeedSetpointFb_Rpm"
   IOField "I/O field_3" at 376,93 size 120x32; FormatPattern s9999.99; Unit  А
      Visibility <- "iVisibilityDevices"
      ProcessValue <- "ActCurrent_A"
   IOField "I/O field_4" at 376,116 size 120x32; FormatPattern s9999.99; Unit  Н*м
      Visibility <- "iVisibilityDevices"
      ProcessValue <- "ActTorque_Nm"
   IOField "I/O field_5" at 376,139 size 120x32; FormatPattern s9999.99; Unit  кВт
      Visibility <- "iVisibilityDevices"
      ProcessValue <- "ActPower_kW"
   IOField "I/O field_6" at 376,162 size 120x32; FormatPattern s9999.99; Unit  %
      Visibility <- "iVisibilityDevices"
      ProcessValue <- "LoadPower_Pct"

